KUKA KRL program: MyProgram_157().src

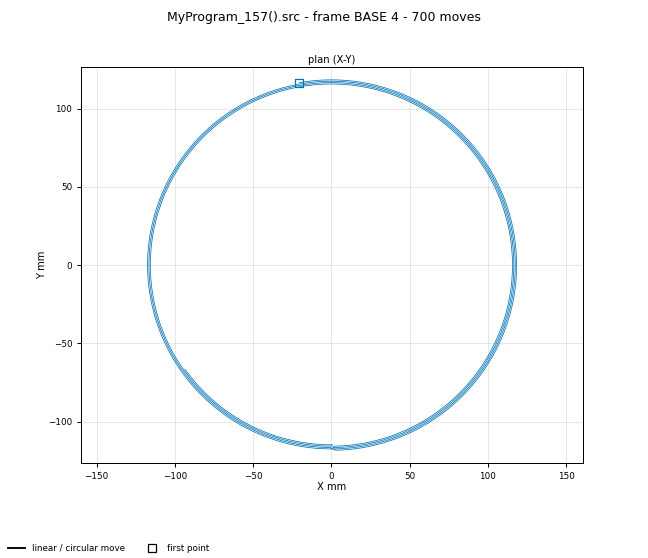
[picture p0: tool path of MyProgram_157().src in frame BASE 4, 700 of 700 moves have a stored position in this frame; points joined in program order, loops and branches not executed]
&ACCESS RVP
&REL 1
&PARAM TEMPLATE = C:\KRC\Roboter\Template\vorgabe
&PARAM EDITMASK = *
DEF MyProgram_157()
; ---- Setting reference (Base) ----
$BASE = BASE_DATA[4]

; --------------------------
; ---- Setting tool (TCP) ----
$TOOL = TOOL_DATA[3]
; --------------------------

$VEL.CP = VEL_APROX_PRINT
Startdeposition()
$VEL.CP = VEL_PRINT
LIN {X -20.7298,Y 116.5177,Z 121,A 95.4648,B 24.939,C -1.8039,E1 24.9731,E2 350.5826} C_DIS
LIN {X -17.3655,Y 117.0684,Z 121,A 93.8121,B 24.939,C -1.8049,E1 24.9777,E2 352.2344} C_DIS
LIN {X -14.6611,Y 117.4368,Z 121,A 92.4805,B 24.939,C -1.8053,E1 24.9814,E2 353.566} C_DIS
LIN {X -10.6565,Y 117.8666,Z 121,A 90.5367,B 24.9388,C -1.8066,E1 24.9868,E2 355.5079} C_DIS
LIN {X -7.2573,Y 118.1266,Z 121,A 88.8847,B 24.9388,C -1.8072,E1 24.9914,E2 357.1591} C_DIS
LIN {X -3.4087,Y 118.2982,Z 121,A 86.9833,B 24.9388,C -1.8062,E1 24.9967,E2 359.0632} C_DIS
LIN {X 0,Y 118.3494,Z 121,A 85.3671,B 24.9388,C -1.8081,E1 25.0012,E2 360.675} C_DIS
LIN {X 2.9044,Y 118.3137,Z 121,A 83.9605,B 24.9388,C -1.8082,E1 25.0051,E2 362.0809} C_DIS
LIN {X 5.8071,Y 118.2068,Z 121,A 82.5537,B 24.9388,C -1.8082,E1 25.009,E2 363.4872} C_DIS
LIN {X 9.9086,Y 117.9326,Z 121,A 80.5481,B 24.9388,C -1.8075,E1 25.0146,E2 365.4936} C_DIS
LIN {X 13.0447,Y 117.6283,Z 121,A 79.0389,B 24.9388,C -1.808,E1 25.0188,E2 367.0007} C_DIS
LIN {X 17.3655,Y 117.0684,Z 121,A 76.9308,B 24.9388,C -1.8076,E1 25.0246,E2 369.1081} C_DIS
LIN {X 21.1661,Y 116.4392,Z 121,A 75.01,B 24.939,C -1.8044,E1 25.0299,E2 371.0343} C_DIS
LIN {X 23.9622,Y 115.896,Z 121,A 73.6209,B 24.939,C -1.8034,E1 25.0338,E2 372.4243} C_DIS
LIN {X 27.3456,Y 115.1468,Z 121,A 72.0133,B 24.9389,C -1.8056,E1 25.0381,E2 374.0244} C_DIS
LIN {X 29.8333,Y 114.5258,Z 121,A 70.7927,B 24.9389,C -1.8058,E1 25.0414,E2 375.2426} C_DIS
LIN {X 32.4772,Y 113.8039,Z 121,A 69.3918,B 24.9392,C -1.8015,E1 25.0452,E2 376.6514} C_DIS
LIN {X 35.2603,Y 112.9726,Z 121,A 67.9878,B 24.9392,C -1.8006,E1 25.0489,E2 378.0551} C_DIS
LIN {X 39.3665,Y 111.608,Z 121,A 65.8909,B 24.9394,C -1.7987,E1 25.0545,E2 380.1524} C_DIS
LIN {X 43.4755,Y 110.0726,Z 121,A 63.8342,B 24.9393,C -1.7996,E1 25.0598,E2 382.2023} C_DIS
LIN {X 46.6287,Y 108.7765,Z 121,A 62.1876,B 24.9394,C -1.798,E1 25.0641,E2 383.8489} C_DIS
LIN {X 49.2842,Y 107.5995,Z 121,A 60.785,B 24.9395,C -1.7965,E1 25.0676,E2 385.2516} C_DIS
LIN {X 52.7592,Y 105.9366,Z 121,A 58.8678,B 24.9398,C -1.7919,E1 25.0725,E2 387.1747} C_DIS
LIN {X 55.7895,Y 104.3748,Z 121,A 57.2788,B 24.9398,C -1.7924,E1 25.0764,E2 388.7579} C_DIS
LIN {X 58.3342,Y 102.9742,Z 121,A 55.877,B 24.9399,C -1.7907,E1 25.0798,E2 390.1599} C_DIS
LIN {X 61.6537,Y 101.0194,Z 121,A 53.9611,B 24.9402,C -1.7855,E1 25.0844,E2 392.0819} C_DIS
LIN {X 64.5389,Y 99.2034,Z 121,A 52.373,B 24.9402,C -1.7858,E1 25.0881,E2 393.6643} C_DIS
LIN {X 67.7323,Y 97.0486,Z 121,A 50.4575,B 24.9406,C -1.7804,E1 25.0926,E2 395.5861} C_DIS
LIN {X 70.303,Y 95.2038,Z 121,A 48.9728,B 24.9406,C -1.7798,E1 25.0959,E2 397.0667} C_DIS
LIN {X 72.8123,Y 93.3003,Z 121,A 47.4695,B 24.9407,C -1.778,E1 25.0992,E2 398.5688} C_DIS
LIN {X 76.1971,Y 90.5571,Z 121,A 45.3689,B 24.941,C -1.7744,E1 25.1038,E2 400.6701} C_DIS
LIN {X 78.3965,Y 88.6598,Z 121,A 43.9683,B 24.9412,C -1.7719,E1 25.1067,E2 402.0711} C_DIS
LIN {X 81.2392,Y 86.0598,Z 121,A 42.1113,B 24.9414,C -1.7684,E1 25.1105,E2 403.9286} C_DIS
LIN {X 83.6856,Y 83.6856,Z 121,A 40.4685,B 24.9416,C -1.7652,E1 25.1138,E2 405.5722} C_DIS
LIN {X 85.7142,Y 81.6067,Z 121,A 39.069,B 24.9418,C -1.7624,E1 25.1165,E2 406.9722} C_DIS
LIN {X 88.6598,Y 78.3965,Z 121,A 36.9698,B 24.9421,C -1.7581,E1 25.1205,E2 409.0723} C_DIS
LIN {X 91.4853,Y 75.08,Z 121,A 34.8712,B 24.9424,C -1.7536,E1 25.1242,E2 411.1719} C_DIS
LIN {X 94.1868,Y 71.6618,Z 121,A 32.7728,B 24.9427,C -1.749,E1 25.1278,E2 413.2714} C_DIS
LIN {X 95.9171,Y 69.3288,Z 121,A 31.3738,B 24.9429,C -1.7458,E1 25.1302,E2 414.6712} C_DIS
LIN {X 97.5896,Y 66.954,Z 121,A 29.9754,B 24.9431,C -1.7426,E1 25.1324,E2 416.0703} C_DIS
LIN {X 99.2034,Y 64.5389,Z 121,A 28.577,B 24.9433,C -1.7393,E1 25.1345,E2 417.4695} C_DIS
LIN {X 100.7574,Y 62.0849,Z 121,A 27.1786,B 24.9435,C -1.7359,E1 25.1366,E2 418.8687} C_DIS
LIN {X 101.9939,Y 60.0278,Z 121,A 25.9667,B 24.9439,C -1.7304,E1 25.1384,E2 420.0873} C_DIS
LIN {X 103.6823,Y 57.0661,Z 121,A 24.3826,B 24.9439,C -1.729,E1 25.1405,E2 421.6666} C_DIS
LIN {X 105.0516,Y 54.5045,Z 121,A 22.9846,B 24.9442,C -1.7255,E1 25.1423,E2 423.0656} C_DIS
LIN {X 106.7681,Y 51.0556,Z 121,A 21.1306,B 24.9445,C -1.7208,E1 25.1446,E2 424.9207} C_DIS
LIN {X 107.9889,Y 48.42,Z 121,A 19.6765,B 24.9449,C -1.7144,E1 25.1463,E2 426.3819} C_DIS
LIN {X 109.3406,Y 45.2903,Z 121,A 18.0929,B 24.945,C -1.7128,E1 25.148,E2 427.9607} C_DIS
LIN {X 110.4191,Y 42.5933,Z 121,A 16.6957,B 24.9453,C -1.709,E1 25.1495,E2 429.359} C_DIS
LIN {X 111.745,Y 38.9763,Z 121,A 14.7858,B 24.9458,C -1.7013,E1 25.1513,E2 431.2764} C_DIS
LIN {X 112.8232,Y 35.7422,Z 121,A 13.2026,B 24.9458,C -1.6995,E1 25.1526,E2 432.8549} C_DIS
LIN {X 113.6663,Y 32.9626,Z 121,A 11.8056,B 24.9461,C -1.6956,E1 25.1537,E2 434.253} C_DIS
LIN {X 114.4411,Y 30.1632,Z 121,A 10.4084,B 24.9464,C -1.6917,E1 25.1548,E2 435.6515} C_DIS
LIN {X 115.1468,Y 27.3456,Z 121,A 9.0115,B 24.9466,C -1.6878,E1 25.1557,E2 437.0495} C_DIS
LIN {X 116.0753,Y 23.0888,Z 121,A 6.9164,B 24.947,C -1.6818,E1 25.1569,E2 439.1465} C_DIS
LIN {X 116.7633,Y 19.2984,Z 121,A 5.0071,B 24.9475,C -1.6738,E1 25.1578,E2 441.0635} C_DIS
LIN {X 117.2017,Y 16.4271,Z 121,A 3.6104,B 24.9478,C -1.6698,E1 25.1584,E2 442.4615} C_DIS
LIN {X 117.5901,Y 13.3702,Z 121,A 2.205,B 24.9478,C -1.6691,E1 25.1589,E2 443.8601} C_DIS
LIN {X 117.8666,Y 10.6565,Z 121,A 0.8739,B 24.9481,C -1.6644,E1 25.1592,E2 445.1945} C_DIS
LIN {X 118.1266,Y 7.2573,Z 121,A -0.7652,B 24.9484,C -1.6595,E1 25.1595,E2 446.8353} C_DIS
LIN {X 118.2982,Y 3.4087,Z 121,A -2.674,B 24.9489,C -1.6514,E1 25.1597,E2 448.7519} C_DIS
LIN {X 118.3493,Y 0,Z 121,A -4.4183,B 24.9495,C -1.6414,E1 25.1597,E2 450.5093} C_DIS
LIN {X 118.2847,Y -3.8518,Z 121,A -6.1653,B 24.9495,C -1.6411,E1 25.1597,E2 452.2467} C_DIS
LIN {X 118.1266,Y -7.2573,Z 121,A -7.7477,B 24.9497,C -1.6389,E1 25.1594,E2 453.8248} C_DIS
LIN {X 117.913,Y -10.1541,Z 121,A -9.1441,B 24.9499,C -1.6348,E1 25.1591,E2 455.2227} C_DIS
LIN {X 117.6283,Y -13.0447,Z 121,A -10.5406,B 24.9502,C -1.6307,E1 25.1587,E2 456.6206} C_DIS
LIN {X 117.0684,Y -17.3655,Z 121,A -12.6352,B 24.9506,C -1.6245,E1 25.1579,E2 458.7174} C_DIS
LIN {X 116.607,Y -20.2332,Z 121,A -14.0318,B 24.9508,C -1.6204,E1 25.1573,E2 460.1155} C_DIS
LIN {X 116.0753,Y -23.0888,Z 121,A -15.4284,B 24.951,C -1.6163,E1 25.1565,E2 461.5137} C_DIS
LIN {X 115.4737,Y -25.9305,Z 121,A -16.825,B 24.9513,C -1.6122,E1 25.1557,E2 462.9117} C_DIS
LIN {X 114.5667,Y -29.6745,Z 121,A -18.6774,B 24.9516,C -1.6068,E1 25.1545,E2 464.766} C_DIS
LIN {X 113.8039,Y -32.4772,Z 121,A -20.1306,B 24.952,C -1.6001,E1 25.1534,E2 466.2269} C_DIS
LIN {X 112.9726,Y -35.2603,Z 121,A -21.5273,B 24.9523,C -1.596,E1 25.1522,E2 467.6251} C_DIS
LIN {X 111.5982,Y -39.3946,Z 121,A -23.6224,B 24.9526,C -1.5901,E1 25.1503,E2 469.7225} C_DIS
LIN {X 110.4191,Y -42.5933,Z 121,A -25.2053,B 24.9527,C -1.5881,E1 25.1488,E2 471.3012} C_DIS
LIN {X 108.7765,Y -46.6287,Z 121,A -27.3008,B 24.9531,C -1.5822,E1 25.1466,E2 473.399} C_DIS
LIN {X 107.8067,Y -48.8242,Z 121,A -28.5117,B 24.9534,C -1.5763,E1 25.1452,E2 474.6172} C_DIS
LIN {X 106.3576,Y -51.91,Z 121,A -30.0949,B 24.9535,C -1.5745,E1 25.1433,E2 476.1962} C_DIS
LIN {X 105.0871,Y -54.4349,Z 121,A -31.4564,B 24.9538,C -1.5708,E1 25.1415,E2 477.5593} C_DIS
LIN {X 103.6823,Y -57.0661,Z 121,A -32.8894,B 24.954,C -1.567,E1 25.1396,E2 478.9938} C_DIS
LIN {X 102.2506,Y -59.5934,Z 121,A -34.287,B 24.9542,C -1.5633,E1 25.1377,E2 480.3928} C_DIS
LIN {X 100.7573,Y -62.0849,Z 121,A -35.6846,B 24.9544,C -1.5596,E1 25.1356,E2 481.792} C_DIS
LIN {X 98.4039,Y -65.7514,Z 121,A -37.7809,B 24.9547,C -1.5542,E1 25.1325,E2 483.8906} C_DIS
LIN {X 96.2101,Y -68.9181,Z 121,A -39.6351,B 24.955,C -1.5495,E1 25.1295,E2 485.7467} C_DIS
LIN {X 94.5528,Y -71.1746,Z 121,A -41.0138,B 24.9553,C -1.5447,E1 25.1272,E2 487.1302} C_DIS
LIN {X 92.3998,Y -73.9517,Z 121,A -42.6739,B 24.9555,C -1.542,E1 25.1243,E2 488.7889} C_DIS
LIN {X 90.5571,Y -76.1971,Z 121,A -44.0724,B 24.9556,C -1.5386,E1 25.1218,E2 490.1888} C_DIS
LIN {X 88.6598,Y -78.3965,Z 121,A -45.4709,B 24.9558,C -1.5353,E1 25.1192,E2 491.5889} C_DIS
LIN {X 86.069,Y -81.2294,Z 121,A -47.3786,B 24.9562,C -1.5283,E1 25.1156,E2 493.5048} C_DIS
LIN {X 83.6856,Y -83.6856,Z 121,A -48.9679,B 24.9562,C -1.5273,E1 25.1125,E2 495.0895} C_DIS
LIN {X 80.9162,Y -86.3635,Z 121,A -50.8798,B 24.9567,C -1.5206,E1 25.1086,E2 497.0094} C_DIS
LIN {X 77.6826,Y -89.2833,Z 121,A -52.9786,B 24.9569,C -1.5162,E1 25.1042,E2 499.1102} C_DIS
LIN {X 74.3437,Y -92.0821,Z 121,A -55.0212,B 24.957,C -1.5146,E1 25.0999,E2 501.1488} C_DIS
LIN {X 72.0615,Y -93.8788,Z 121,A -56.4774,B 24.9573,C -1.5091,E1 25.0966,E2 502.6125} C_DIS
LIN {X 69.3288,Y -95.9171,Z 121,A -58.0641,B 24.9573,C -1.5086,E1 25.0931,E2 504.1947} C_DIS
LIN {X 66.954,Y -97.5896,Z 121,A -59.4641,B 24.9575,C -1.506,E1 25.0899,E2 505.5961} C_DIS
LIN {X 64.9601,Y -98.9256,Z 121,A -60.6777,B 24.9578,C -1.5013,E1 25.087,E2 506.8168} C_DIS
LIN {X 62.0849,Y -100.7573,Z 121,A -62.2646,B 24.9578,C -1.5011,E1 25.0833,E2 508.3991} C_DIS
LIN {X 59.5934,Y -102.2506,Z 121,A -63.6655,B 24.9579,C -1.4987,E1 25.0799,E2 509.8013} C_DIS
LIN {X 56.233,Y -104.1343,Z 121,A -65.4978,B 24.958,C -1.497,E1 25.0754,E2 511.6324} C_DIS
LIN {X 53.6605,Y -105.4829,Z 121,A -66.9246,B 24.9582,C -1.4936,E1 25.0719,E2 513.0632} C_DIS
LIN {X 51.0556,Y -106.7681,Z 121,A -68.3222,B 24.9583,C -1.4917,E1 25.0684,E2 514.4616} C_DIS
LIN {X 47.9601,Y -108.1961,Z 121,A -69.9709,B 24.9585,C -1.4892,E1 25.0642,E2 516.1122} C_DIS
LIN {X 43.9452,Y -109.8881,Z 121,A -72.0737,B 24.9586,C -1.4864,E1 25.0587,E2 518.2167} C_DIS
LIN {X 40.3447,Y -111.2583,Z 121,A -73.9903,B 24.9589,C -1.4815,E1 25.0537,E2 520.1408} C_DIS
LIN {X 36.2222,Y -112.6678,Z 121,A -76.0939,B 24.959,C -1.4791,E1 25.0481,E2 522.246} C_DIS
LIN {X 33.4463,Y -113.5229,Z 121,A -77.4966,B 24.959,C -1.4777,E1 25.0444,E2 523.6497} C_DIS
LIN {X 30.1632,Y -114.4411,Z 121,A -79.0867,B 24.959,C -1.4786,E1 25.0401,E2 525.2349} C_DIS
LIN {X 26.4221,Y -115.3602,Z 121,A -80.9477,B 24.9591,C -1.477,E1 25.0351,E2 527.0971} C_DIS
LIN {X 23.0888,Y -116.0753,Z 121,A -82.5949,B 24.9592,C -1.4757,E1 25.0306,E2 528.7454} C_DIS
LIN {X 19.2984,Y -116.7633,Z 121,A -84.5139,B 24.9594,C -1.4717,E1 25.0253,E2 530.6717} C_DIS
LIN {X 16.4271,Y -117.2017,Z 121,A -85.9181,B 24.9594,C -1.4708,E1 25.0214,E2 532.0767} C_DIS
LIN {X 13.0447,Y -117.6283,Z 121,A -87.5095,B 24.9594,C -1.4725,E1 25.017,E2 533.663} C_DIS
LIN {X 10.1541,Y -117.913,Z 121,A -88.9137,B 24.9594,C -1.4718,E1 25.0131,E2 535.0679} C_DIS
LIN {X 7.2573,Y -118.1266,Z 121,A -90.3189,B 24.9594,C -1.4712,E1 25.0092,E2 536.4739} C_DIS
LIN {X 2.9044,Y -118.3137,Z 121,A -92.4266,B 24.9594,C -1.4706,E1 25.0033,E2 538.5826} C_DIS
LIN {X 2.9044,Y -118.3137,Z 121,A -92.4266,B 24.9594,C -1.4706,E1 25.0033,E2 538.5826} C_DIS
Enddeposition()
LIN {X 0.8321,Y -117.4596,Z 121,A -93.3395,B 24.9584,C -1.49,E1 25.0009,E2 539.4494} C_DIS
Startdeposition()
$VEL.CP = VEL_PRINT
LIN {X 3.2999,Y -117.4195,Z 121,A -91.5559,B 24.9569,C -1.5166,E1 25.006,E2 537.603} C_DIS
LIN {X 6.8139,Y -117.2681,Z 121,A -89.8243,B 24.9569,C -1.518,E1 25.0108,E2 535.8686} C_DIS
LIN {X 10.3893,Y -117.0058,Z 121,A -88.0253,B 24.9566,C -1.5212,E1 25.0159,E2 534.0631} C_DIS
LIN {X 14.3068,Y -116.5927,Z 121,A -86.0792,B 24.9566,C -1.5235,E1 25.0213,E2 532.1131} C_DIS
LIN {X 17.0501,Y -116.2227,Z 121,A -84.8996,B 24.9569,C -1.5166,E1 25.0245,E2 530.9508} C_DIS
LIN {X 21.5545,Y -115.4729,Z 121,A -82.5382,B 24.9565,C -1.5245,E1 25.031,E2 528.5731} C_DIS
LIN {X 24.947,Y -114.7858,Z 121,A -80.9226,B 24.9565,C -1.5227,E1 25.0354,E2 526.964} C_DIS
LIN {X 27.5735,Y -114.1837,Z 121,A -79.0122,B 24.9549,C -1.5518,E1 25.0408,E2 524.9874} C_DIS
LIN {X 31.8685,Y -113.06,Z 121,A -77.3966,B 24.9562,C -1.5284,E1 25.045,E2 523.4297} C_DIS
LIN {X 36.1496,Y -111.7647,Z 121,A -75.3333,B 24.9564,C -1.5255,E1 25.0505,E2 521.3772} C_DIS
LIN {X 39.0961,Y -110.7685,Z 121,A -73.7738,B 24.9562,C -1.5294,E1 25.0546,E2 519.8115} C_DIS
LIN {X 43.4706,Y -109.1272,Z 121,A -71.4393,B 24.9558,C -1.5351,E1 25.0607,E2 517.4685} C_DIS
LIN {X 46.5849,Y -107.8338,Z 121,A -69.8145,B 24.9558,C -1.5366,E1 25.0649,E2 515.844} C_DIS
LIN {X 49.5604,Y -106.4984,Z 121,A -68.2686,B 24.9558,C -1.537,E1 25.0688,E2 514.301} C_DIS
LIN {X 53.0811,Y -104.7889,Z 121,A -66.5543,B 24.9561,C -1.531,E1 25.073,E2 512.6055} C_DIS
LIN {X 56.616,Y -102.9234,Z 121,A -64.3099,B 24.9551,C -1.5483,E1 25.0786,E2 510.3266} C_DIS
LIN {X 59.527,Y -101.2657,Z 121,A -62.7876,B 24.9552,C -1.546,E1 25.0823,E2 508.8144} C_DIS
LIN {X 62.3026,Y -99.5818,Z 121,A -61.1934,B 24.955,C -1.5496,E1 25.0861,E2 507.2167} C_DIS
LIN {X 65.7863,Y -97.3155,Z 121,A -59.2186,B 24.955,C -1.5511,E1 25.0907,E2 505.2449} C_DIS
LIN {X 68.4047,Y -95.4933,Z 121,A -57.8037,B 24.9551,C -1.5477,E1 25.0939,E2 503.8431} C_DIS
LIN {X 72.3765,Y -92.5208,Z 121,A -54.5882,B 24.9526,C -1.591,E1 25.1012,E2 500.5371} C_DIS
LIN {X 75.9705,Y -89.5918,Z 121,A -52.9888,B 24.9542,C -1.5643,E1 25.1045,E2 499.0069} C_DIS
LIN {X 79.7422,Y -86.2515,Z 121,A -50.3792,B 24.9534,C -1.5774,E1 25.1099,E2 496.3768} C_DIS
LIN {X 83.2682,Y -82.8525,Z 121,A -47.8356,B 24.9526,C -1.5907,E1 25.115,E2 493.8125} C_DIS
LIN {X 85.5139,Y -80.5327,Z 121,A -46.7222,B 24.9537,C -1.5725,E1 25.1171,E2 492.7469} C_DIS
LIN {X 88.3698,Y -77.3882,Z 121,A -44.5319,B 24.953,C -1.5835,E1 25.1212,E2 490.5404} C_DIS
LIN {X 90.7856,Y -74.5426,Z 121,A -42.7886,B 24.953,C -1.5845,E1 25.1243,E2 488.8026} C_DIS
LIN {X 92.9303,Y -71.848,Z 121,A -41.0839,B 24.9526,C -1.5903,E1 25.1272,E2 487.0923} C_DIS
LIN {X 94.8498,Y -69.2941,Z 121,A -39.5118,B 24.9523,C -1.5953,E1 25.1299,E2 485.516} C_DIS
LIN {X 97.0567,Y -66.1684,Z 121,A -37.7561,B 24.9523,C -1.5952,E1 25.1326,E2 483.7692} C_DIS
LIN {X 98.672,Y -63.7345,Z 121,A -36.434,B 24.9523,C -1.5943,E1 25.1347,E2 482.4557} C_DIS
LIN {X 100.7204,Y -60.448,Z 121,A -34.2239,B 24.9511,C -1.6153,E1 25.1379,E2 480.2075} C_DIS
LIN {X 102.8049,Y -56.829,Z 121,A -32.2704,B 24.951,C -1.6172,E1 25.1406,E2 478.2595} C_DIS
LIN {X 104.4904,Y -53.6651,Z 121,A -30.6953,B 24.9512,C -1.6141,E1 25.1426,E2 476.7001} C_DIS
LIN {X 105.8226,Y -50.9876,Z 121,A -29.2209,B 24.9509,C -1.6193,E1 25.1444,E2 475.2214} C_DIS
LIN {X 107.3121,Y -47.7758,Z 121,A -27.3557,B 24.9501,C -1.6312,E1 25.1466,E2 473.3381} C_DIS
LIN {X 108.8767,Y -44.0914,Z 121,A -25.4954,B 24.9501,C -1.6328,E1 25.1486,E2 471.4843} C_DIS
LIN {X 110.3331,Y -40.3081,Z 121,A -23.5273,B 24.9497,C -1.6386,E1 25.1505,E2 469.5135} C_DIS
LIN {X 112.5098,Y -33.7612,Z 121,A -20.1836,B 24.9491,C -1.6482,E1 25.1534,E2 466.1663} C_DIS
LIN {X 113.818,Y -29.0452,Z 121,A -17.8234,B 24.9487,C -1.6545,E1 25.1551,E2 463.8046} C_DIS
LIN {X 114.7059,Y -25.3135,Z 121,A -15.9774,B 24.9484,C -1.6593,E1 25.1563,E2 461.958} C_DIS
LIN {X 115.4119,Y -21.8711,Z 121,A -14.3015,B 24.9482,C -1.663,E1 25.1572,E2 460.2832} C_DIS
LIN {X 115.9573,Y -18.7721,Z 121,A -12.6525,B 24.9475,C -1.6736,E1 25.158,E2 458.619} C_DIS
LIN {X 116.5771,Y -14.4341,Z 121,A -10.4812,B 24.947,C -1.6822,E1 25.1588,E2 456.4402} C_DIS
LIN {X 116.9803,Y -10.6656,Z 121,A -8.7611,B 24.947,C -1.682,E1 25.1592,E2 454.7308} C_DIS
LIN {X 117.2798,Y -6.603,Z 121,A -6.7288,B 24.9464,C -1.6907,E1 25.1596,E2 452.6899} C_DIS
LIN {X 117.4395,Y -2.4929,Z 121,A -4.8179,B 24.9464,C -1.6926,E1 25.1598,E2 450.7859} C_DIS
LIN {X 117.4621,Y 0.9671,Z 121,A -3.0388,B 24.9457,C -1.7026,E1 25.1598,E2 448.994} C_DIS
LIN {X 117.3604,Y 4.967,Z 121,A -1.1861,B 24.9456,C -1.7041,E1 25.1596,E2 447.1487} C_DIS
LIN {X 117.1297,Y 8.8879,Z 121,A 0.6551,B 24.9454,C -1.7067,E1 25.1592,E2 445.3123} C_DIS
LIN {X 116.8294,Y 12.2075,Z 121,A 2.3671,B 24.9448,C -1.7161,E1 25.1588,E2 443.5882} C_DIS
LIN {X 116.3353,Y 16.2574,Z 121,A 4.3009,B 24.9446,C -1.7198,E1 25.1581,E2 441.6572} C_DIS
LIN {X 115.8422,Y 19.4608,Z 121,A 5.83,B 24.9444,C -1.7223,E1 25.1574,E2 440.1311} C_DIS
LIN {X 115.2313,Y 22.8093,Z 121,A 7.8143,B 24.943,C -1.7432,E1 25.1563,E2 438.1091} C_DIS
LIN {X 114.1359,Y 27.7692,Z 121,A 9.9681,B 24.9436,C -1.7353,E1 25.155,E2 435.9864} C_DIS
LIN {X 113.2965,Y 31.0193,Z 121,A 11.5935,B 24.9433,C -1.7398,E1 25.1538,E2 434.3598} C_DIS
LIN {X 112.537,Y 33.6693,Z 121,A 13.2708,B 24.9419,C -1.76,E1 25.1525,E2 432.6443} C_DIS
LIN {X 111.5369,Y 36.8533,Z 121,A 14.6663,B 24.9424,C -1.7537,E1 25.1513,E2 431.2717} C_DIS
LIN {X 110.3661,Y 40.2178,Z 121,A 16.2948,B 24.9424,C -1.7537,E1 25.1497,E2 429.6524} C_DIS
LIN {X 108.9824,Y 43.8315,Z 121,A 18.1047,B 24.9422,C -1.7555,E1 25.1479,E2 427.8482} C_DIS
LIN {X 107.6921,Y 46.91,Z 121,A 19.6476,B 24.9422,C -1.7562,E1 25.1462,E2 426.3122} C_DIS
LIN {X 106.1333,Y 50.3408,Z 121,A 22.3438,B 24.9391,C -1.8028,E1 25.1429,E2 423.5204} C_DIS
LIN {X 103.8916,Y 54.815,Z 121,A 24.0413,B 24.941,C -1.7738,E1 25.1408,E2 421.9004} C_DIS
LIN {X 102.0703,Y 58.1377,Z 121,A 25.8931,B 24.9407,C -1.779,E1 25.1383,E2 420.0459} C_DIS
LIN {X 100.5204,Y 60.777,Z 121,A 27.2357,B 24.9409,C -1.7759,E1 25.1364,E2 418.7176} C_DIS
LIN {X 98.6915,Y 63.7041,Z 121,A 29.5071,B 24.9387,C -1.8085,E1 25.1329,E2 416.3808} C_DIS
LIN {X 96.5397,Y 66.9196,Z 121,A 31.326,B 24.9386,C -1.81,E1 25.13,E2 414.5671} C_DIS
LIN {X 94.3656,Y 69.9551,Z 121,A 32.6495,B 24.9399,C -1.7908,E1 25.1279,E2 413.2954} C_DIS
LIN {X 92.4451,Y 72.4724,Z 121,A 34.2293,B 24.9395,C -1.7963,E1 25.1252,E2 411.7102} C_DIS
LIN {X 90.7782,Y 74.5514,Z 121,A 35.6238,B 24.939,C -1.8039,E1 25.1227,E2 410.3042} C_DIS
LIN {X 88.4019,Y 77.3515,Z 121,A 37.3344,B 24.939,C -1.8043,E1 25.1196,E2 408.6004} C_DIS
LIN {X 85.9021,Y 80.1199,Z 121,A 39.2627,B 24.9384,C -1.8135,E1 25.1159,E2 406.6587} C_DIS
LIN {X 82.9142,Y 83.2084,Z 121,A 41.2151,B 24.9385,C -1.8113,E1 25.1121,E2 404.7199} C_DIS
LIN {X 80.6743,Y 85.3807,Z 121,A 42.7029,B 24.9384,C -1.8129,E1 25.1091,E2 403.2344} C_DIS
LIN {X 78.2297,Y 87.6258,Z 121,A 44.343,B 24.9381,C -1.8172,E1 25.1057,E2 401.5908} C_DIS
LIN {X 75.253,Y 90.1952,Z 121,A 46.9929,B 24.9355,C -1.8554,E1 25.0999,E2 398.8607} C_DIS
LIN {X 71.2921,Y 93.3586,Z 121,A 48.8424,B 24.9372,C -1.8306,E1 25.0959,E2 397.0768} C_DIS
LIN {X 68.8181,Y 95.1982,Z 121,A 50.3454,B 24.937,C -1.8332,E1 25.0926,E2 395.573} C_DIS
LIN {X 66.325,Y 96.9508,Z 121,A 51.7855,B 24.937,C -1.8335,E1 25.0892,E2 394.137} C_DIS
LIN {X 63.5754,Y 98.7741,Z 121,A 53.1884,B 24.9375,C -1.8265,E1 25.086,E2 392.7552} C_DIS
LIN {X 61.2629,Y 100.2251,Z 121,A 54.5665,B 24.9372,C -1.8308,E1 25.0827,E2 391.3715} C_DIS
LIN {X 58.2969,Y 101.9788,Z 121,A 56.3672,B 24.9366,C -1.8388,E1 25.0783,E2 389.5572} C_DIS
LIN {X 54.7673,Y 103.9167,Z 121,A 58.3102,B 24.9366,C -1.8405,E1 25.0736,E2 387.6157} C_DIS
LIN {X 51.2509,Y 105.696,Z 121,A 60.2593,B 24.9363,C -1.8442,E1 25.0687,E2 385.6632} C_DIS
LIN {X 47.6547,Y 107.3667,Z 121,A 62.1737,B 24.9362,C -1.8455,E1 25.0638,E2 383.7505} C_DIS
LIN {X 44.4763,Y 108.72,Z 121,A 63.8325,B 24.9362,C -1.8461,E1 25.0596,E2 382.0941} C_DIS
LIN {X 40.8745,Y 110.1265,Z 121,A 65.7701,B 24.9358,C -1.8503,E1 25.0545,E2 380.1508} C_DIS
LIN {X 37.3056,Y 111.3844,Z 121,A 68.0183,B 24.9344,C -1.8703,E1 25.0484,E2 377.8594} C_DIS
LIN {X 33.5434,Y 112.5744,Z 121,A 69.8704,B 24.9346,C -1.8684,E1 25.0435,E2 376.0151} C_DIS
LIN {X 29.9249,Y 113.5918,Z 121,A 71.2033,B 24.9361,C -1.8468,E1 25.04,E2 374.7356} C_DIS
LIN {X 26.9203,Y 114.3402,Z 121,A 72.8671,B 24.9355,C -1.8546,E1 25.0355,E2 373.0557} C_DIS
LIN {X 23.1374,Y 115.1653,Z 121,A 74.7881,B 24.9354,C -1.857,E1 25.0302,E2 371.1314} C_DIS
LIN {X 19.1105,Y 115.9008,Z 121,A 76.6553,B 24.9357,C -1.8519,E1 25.0251,E2 369.2784} C_DIS
LIN {X 15.7309,Y 116.4091,Z 121,A 78.2397,B 24.9359,C -1.8486,E1 25.0208,E2 367.7031} C_DIS
LIN {X 12.4103,Y 116.8082,Z 121,A 79.9364,B 24.9357,C -1.8518,E1 25.016,E2 365.9999} C_DIS
LIN {X 9.0609,Y 117.1159,Z 121,A 81.691,B 24.9354,C -1.8571,E1 25.0111,E2 364.2339} C_DIS
LIN {X 5.751,Y 117.3267,Z 121,A 83.3791,B 24.9351,C -1.8601,E1 25.0064,E2 362.5391} C_DIS
LIN {X 1.4546,Y 117.4582,Z 121,A 85.3149,B 24.9357,C -1.8527,E1 25.001,E2 360.6213} C_DIS
LIN {X -1.9991,Y 117.4486,Z 121,A 87.0648,B 24.9355,C -1.8553,E1 24.9961,E2 358.8653} C_DIS
LIN {X -6.0792,Y 117.3087,Z 121,A 88.8438,B 24.9362,C -1.8452,E1 24.9912,E2 357.1098} C_DIS
LIN {X -8.9147,Y 117.1275,Z 121,A 90.2049,B 24.9362,C -1.8435,E1 24.9875,E2 355.7522} C_DIS
LIN {X -12.0639,Y 116.8444,Z 121,A 91.9415,B 24.9358,C -1.8513,E1 24.9826,E2 353.9961} C_DIS
LIN {X -15.7391,Y 116.4081,Z 121,A 93.8439,B 24.9355,C -1.8545,E1 24.9773,E2 352.0849} C_DIS
LIN {X -19.8135,Y 115.7832,Z 121,A 95.9275,B 24.9355,C -1.8562,E1 24.9715,E2 349.9951} C_DIS
LIN {X -27.3101,Y 114.2476,Z 121,A 99.7512,B 24.9354,C -1.8569,E1 24.9611,E2 346.1651} C_DIS
LIN {X -32.0342,Y 113.013,Z 121,A 101.8923,B 24.9363,C -1.8439,E1 24.9554,E2 344.0515} C_DIS
LIN {X -35.7831,Y 111.8832,Z 121,A 103.8824,B 24.9362,C -1.8452,E1 24.9501,E2 342.055} C_DIS
LIN {X -39.636,Y 110.5783,Z 121,A 105.7936,B 24.9366,C -1.8395,E1 24.945,E2 340.1535} C_DIS
LIN {X -43.2643,Y 109.2083,Z 121,A 107.6527,B 24.9368,C -1.8356,E1 24.9402,E2 338.2999} C_DIS
LIN {X -50.1091,Y 106.243,Z 121,A 111.442,B 24.9368,C -1.8365,E1 24.9305,E2 334.4992} C_DIS
LIN {X -52.5867,Y 105.0381,Z 121,A 112.9317,B 24.9365,C -1.8406,E1 24.9268,E2 332.9958} C_DIS
LIN {X -56.8256,Y 102.8068,Z 121,A 115.0146,B 24.9375,C -1.8257,E1 24.9217,E2 330.9425} C_DIS
LIN {X -59.2175,Y 101.4487,Z 121,A 116.4587,B 24.9374,C -1.8277,E1 24.9182,E2 329.4895} C_DIS
LIN {X -62.1676,Y 99.6661,Z 121,A 117.9064,B 24.9383,C -1.8146,E1 24.9148,E2 328.0684} C_DIS
LIN {X -64.0959,Y 98.4392,Z 121,A 119.288,B 24.9377,C -1.8238,E1 24.9115,E2 326.6604} C_DIS
LIN {X -68.4041,Y 95.4938,Z 121,A 121.8034,B 24.9381,C -1.8174,E1 24.9058,E2 324.1518} C_DIS
LIN {X -71.4545,Y 93.2335,Z 121,A 123.6221,B 24.9385,C -1.812,E1 24.9017,E2 322.3392} C_DIS
LIN {X -74.1517,Y 91.1028,Z 121,A 125.3091,B 24.9387,C -1.8088,E1 24.8981,E2 320.6536} C_DIS
LIN {X -77.1304,Y 88.595,Z 121,A 127.0055,B 24.9395,C -1.7959,E1 24.8945,E2 318.9812} C_DIS
LIN {X -79.3821,Y 86.583,Z 121,A 128.6575,B 24.9393,C -1.8,E1 24.891,E2 317.3128} C_DIS
LIN {X -82.1034,Y 84.0093,Z 121,A 130.5775,B 24.9393,C -1.7996,E1 24.8872,E2 315.386} C_DIS
LIN {X -84.7278,Y 81.3595,Z 121,A 132.3892,B 24.9396,C -1.7948,E1 24.8836,E2 313.5779} C_DIS
LIN {X -87.3955,Y 78.4869,Z 121,A 134.2484,B 24.9401,C -1.7877,E1 24.8802,E2 311.7273} C_DIS
LIN {X -89.7973,Y 75.7293,Z 121,A 136.0212,B 24.9404,C -1.7826,E1 24.8769,E2 309.9586} C_DIS
LIN {X -92.094,Y 72.9167,Z 121,A 137.7038,B 24.941,C -1.7742,E1 24.874,E2 308.2882} C_DIS
LIN {X -93.5149,Y 71.0883,Z 121,A 139.1211,B 24.9404,C -1.7831,E1 24.8716,E2 306.8428} C_DIS
LIN {X -95.6872,Y 68.1329,Z 121,A 140.7571,B 24.9412,C -1.7718,E1 24.8689,E2 305.2258} C_DIS
LIN {X -97.8621,Y 64.9713,Z 121,A 142.6397,B 24.9415,C -1.767,E1 24.866,E2 303.3453} C_DIS
LIN {X -99.5406,Y 62.3684,Z 121,A 144.1789,B 24.9417,C -1.7639,E1 24.8637,E2 301.8057} C_DIS
LIN {X -101.396,Y 59.3066,Z 121,A 146.0219,B 24.9417,C -1.7628,E1 24.861,E2 299.9557} C_DIS
LIN {X -103.6755,Y 55.2253,Z 121,A 148.2584,B 24.9423,C -1.7543,E1 24.8581,E2 297.7279} C_DIS
LIN {X -104.8636,Y 52.9348,Z 121,A 149.7413,B 24.942,C -1.7598,E1 24.8562,E2 296.2237} C_DIS
LIN {X -106.9367,Y 48.6088,Z 121,A 151.6356,B 24.9436,C -1.7343,E1 24.854,E2 294.3801} C_DIS
LIN {X -108.0879,Y 45.9925,Z 121,A 153.058,B 24.9438,C -1.7311,E1 24.8524,E2 292.9573} C_DIS
LIN {X -109.2054,Y 43.2716,Z 121,A 154.6453,B 24.9438,C -1.733,E1 24.8507,E2 291.3566} C_DIS
LIN {X -110.2298,Y 40.5914,Z 121,A 156.0709,B 24.9439,C -1.7297,E1 24.8493,E2 289.9309} C_DIS
LIN {X -111.4801,Y 37.0217,Z 121,A 158.1326,B 24.9437,C -1.7329,E1 24.8474,E2 287.8499} C_DIS
LIN {X -112.7909,Y 32.8137,Z 121,A 160.2245,B 24.9443,C -1.7237,E1 24.8458,E2 285.7679} C_DIS
LIN {X -114.6039,Y 25.7787,Z 121,A 163.7731,B 24.945,C -1.7124,E1 24.8434,E2 282.2253} C_DIS
LIN {X -115.3539,Y 22.1723,Z 121,A 165.3692,B 24.9459,C -1.6984,E1 24.8425,E2 280.6533} C_DIS
LIN {X -116.0063,Y 18.4644,Z 121,A 167.4636,B 24.9456,C -1.7031,E1 24.8415,E2 278.5353} C_DIS
LIN {X -116.5625,Y 14.5472,Z 121,A 169.2381,B 24.9465,C -1.6904,E1 24.8409,E2 276.7805} C_DIS
LIN {X -116.9389,Y 11.1147,Z 121,A 170.9896,B 24.9466,C -1.6877,E1 24.8404,E2 275.025} C_DIS
LIN {X -117.2413,Y 7.2822,Z 121,A 172.9883,B 24.9466,C -1.6866,E1 24.84,E2 273.0166} C_DIS
LIN {X -117.4349,Y 2.7421,Z 121,A 175.3055,B 24.9469,C -1.6836,E1 24.8398,E2 270.6928} C_DIS
LIN {X -117.4508,Y -1.8747,Z 121,A 177.3802,B 24.9478,C -1.6689,E1 24.8398,E2 268.6405} C_DIS
LIN {X -117.3633,Y -4.8994,Z 121,A 178.8763,B 24.9481,C -1.665,E1 24.84,E2 267.1449} C_DIS
LIN {X -117.1316,Y -8.8645,Z 121,A -179.1565,B 24.9484,C -1.6599,E1 24.8403,E2 265.1778} C_DIS
LIN {X -116.8302,Y -12.1999,Z 121,A -177.574,B 24.9488,C -1.6526,E1 24.8408,E2 263.6034} C_DIS
LIN {X -116.453,Y -15.3921,Z 121,A -176.112,B 24.9494,C -1.6432,E1 24.8413,E2 262.1551} C_DIS
LIN {X -115.7092,Y -20.244,Z 121,A -173.4721,B 24.9492,C -1.6457,E1 24.8425,E2 259.4935} C_DIS
LIN {X -114.6123,Y -25.7423,Z 121,A -170.7012,B 24.9497,C -1.6386,E1 24.844,E2 256.7232} C_DIS
LIN {X -113.8328,Y -28.9879,Z 121,A -169.2105,B 24.9503,C -1.6278,E1 24.845,E2 255.2494} C_DIS
LIN {X -113.1263,Y -31.6345,Z 121,A -167.8365,B 24.9505,C -1.6253,E1 24.846,E2 253.8734} C_DIS
LIN {X -112.1911,Y -34.8035,Z 121,A -166.194,B 24.9507,C -1.6217,E1 24.8474,E2 252.2302} C_DIS
LIN {X -110.9879,Y -38.471,Z 121,A -164.1531,B 24.9507,C -1.6226,E1 24.8492,E2 250.1754} C_DIS
LIN {X -109.5191,Y -42.4731,Z 121,A -162.354,B 24.9518,C -1.6047,E1 24.8509,E2 248.4089} C_DIS
LIN {X -108.6609,Y -44.6215,Z 121,A -160.7538,B 24.9508,C -1.6212,E1 24.8527,E2 246.7604} C_DIS
LIN {X -107.396,Y -47.5891,Z 121,A -159.361,B 24.9515,C -1.609,E1 24.8542,E2 245.389} C_DIS
LIN {X -105.5624,Y -51.5289,Z 121,A -157.2238,B 24.9518,C -1.6037,E1 24.8568,E2 243.2528} C_DIS
LIN {X -104.0752,Y -54.4664,Z 121,A -155.6677,B 24.9522,C -1.5971,E1 24.8588,E2 241.704} C_DIS
LIN {X -102.3643,Y -57.6181,Z 121,A -153.9344,B 24.9525,C -1.5917,E1 24.8611,E2 239.9747} C_DIS
LIN {X -100.4968,Y -60.816,Z 121,A -152.1361,B 24.9528,C -1.5865,E1 24.8637,E2 238.1794} C_DIS
LIN {X -98.7032,Y -63.6859,Z 121,A -150.4671,B 24.9531,C -1.5829,E1 24.8662,E2 236.5105} C_DIS
LIN {X -96.0864,Y -67.5718,Z 121,A -148.0928,B 24.9531,C -1.5808,E1 24.87,E2 234.1294} C_DIS
LIN {X -93.3646,Y -71.2843,Z 121,A -145.8212,B 24.9534,C -1.5764,E1 24.8738,E2 231.8574} C_DIS
LIN {X -90.7928,Y -74.5339,Z 121,A -143.7589,B 24.9536,C -1.5733,E1 24.8774,E2 229.7929} C_DIS
LIN {X -88.1642,Y -77.6236,Z 121,A -141.8114,B 24.954,C -1.5674,E1 24.8809,E2 227.8506} C_DIS
LIN {X -85.4616,Y -80.5883,Z 121,A -139.9323,B 24.9544,C -1.5597,E1 24.8845,E2 225.9816} C_DIS
LIN {X -82.0192,Y -84.092,Z 121,A -137.4604,B 24.9545,C -1.5578,E1 24.8894,E2 223.5038} C_DIS
LIN {X -79.3648,Y -86.5989,Z 121,A -135.7582,B 24.9549,C -1.5508,E1 24.8929,E2 221.8113} C_DIS
LIN {X -76.776,Y -88.9045,Z 121,A -134.1143,B 24.9553,C -1.5454,E1 24.8963,E2 220.1737} C_DIS
LIN {X -73.5801,Y -91.5661,Z 121,A -131.9406,B 24.9551,C -1.5478,E1 24.901,E2 217.986} C_DIS
LIN {X -70.7046,Y -93.8031,Z 121,A -130.3748,B 24.9558,C -1.5355,E1 24.9044,E2 216.4438} C_DIS
LIN {X -68.7447,Y -95.2506,Z 121,A -128.9388,B 24.9553,C -1.5441,E1 24.9077,E2 214.9822} C_DIS
LIN {X -65.7672,Y -97.3284,Z 121,A -127.2548,B 24.9557,C -1.5375,E1 24.9116,E2 213.3084} C_DIS
LIN {X -62.7507,Y -99.3018,Z 121,A -125.4017,B 24.9557,C -1.5388,E1 24.916,E2 211.4462} C_DIS
LIN {X -60.0157,Y -100.9769,Z 121,A -123.952,B 24.9561,C -1.5315,E1 24.9194,E2 210.0094} C_DIS
LIN {X -57.3493,Y -102.5144,Z 121,A -122.337,B 24.9559,C -1.5344,E1 24.9234,E2 208.3829} C_DIS
LIN {X -53.8792,Y -104.381,Z 121,A -120.4191,B 24.956,C -1.5317,E1 24.9281,E2 206.4662} C_DIS
LIN {X -50.3124,Y -106.147,Z 121,A -118.4435,B 24.956,C -1.5308,E1 24.9331,E2 204.4874} C_DIS
LIN {X -47.009,Y -107.6489,Z 121,A -116.7275,B 24.9563,C -1.5265,E1 24.9374,E2 202.7777} C_DIS
LIN {X -43.1896,Y -109.2376,Z 121,A -114.75,B 24.9566,C -1.5226,E1 24.9425,E2 200.8048} C_DIS
LIN {X -40.4795,Y -110.2706,Z 121,A -112.0472,B 24.9533,C -1.5792,E1 24.9501,E2 197.9624} C_DIS
LIN {X -33.287,Y -112.6505,Z 121,A -109.9414,B 24.9576,C -1.5049,E1 24.9552,E2 196.0292} C_DIS
LIN {X -29.9898,Y -113.5746,Z 121,A -107.8447,B 24.9566,C -1.5228,E1 24.9609,E2 193.8868} C_DIS
LIN {X -26.3643,Y -114.4686,Z 121,A -106.1706,B 24.957,C -1.5153,E1 24.9654,E2 192.2283} C_DIS
LIN {X -23.0894,Y -115.1751,Z 121,A -104.4831,B 24.9569,C -1.5169,E1 24.9701,E2 190.5348} C_DIS
LIN {X -20.1568,Y -115.7249,Z 121,A -103.0811,B 24.9571,C -1.514,E1 24.9739,E2 189.1383} C_DIS
LIN {X -16.6179,Y -116.2841,Z 121,A -101.3363,B 24.9571,C -1.5135,E1 24.9787,E2 187.3934} C_DIS
LIN {X -13.4337,Y -116.695,Z 121,A -99.7072,B 24.9569,C -1.5161,E1 24.9833,E2 185.757} C_DIS
LIN {X -9.6354,Y -117.0699,Z 121,A -97.9044,B 24.9571,C -1.5133,E1 24.9883,E2 183.9599} C_DIS
LIN {X -6.2546,Y -117.299,Z 121,A -96.2283,B 24.9571,C -1.5144,E1 24.9929,E2 182.2806} C_DIS
LIN {X -2.1973,Y -117.4449,Z 121,A -94.2612,B 24.9571,C -1.5141,E1 24.9984,E2 180.3141} C_DIS
LIN {X 0.8321,Y -117.4596,Z 121,A -93.3379,B 24.9584,C -1.4893,E1 25.0009,E2 179.4494} C_DIS
Enddeposition()
LIN {X 0.8321,Y -117.4596,Z 121,A -93.3379,B 24.9584,C -1.4893,E1 25.0009,E2 179.4494} C_DIS
Startdeposition()
$VEL.CP = VEL_PRINT
LIN {X -0.7505,Y -116.5814,Z 121,A -94.3235,B 24.9581,C -1.4953,E1 24.9981,E2 180.4208} C_DIS
LIN {X -4.6276,Y -116.4925,Z 121,A -96.2469,B 24.9581,C -1.4943,E1 24.9928,E2 182.3469} C_DIS
LIN {X -7.9922,Y -116.3096,Z 121,A -97.8524,B 24.9581,C -1.4965,E1 24.9883,E2 183.9478} C_DIS
LIN {X -11.7385,Y -115.992,Z 121,A -99.7788,B 24.9582,C -1.4931,E1 24.9829,E2 185.8831} C_DIS
LIN {X -15.2044,Y -115.5883,Z 121,A -101.8987,B 24.9592,C -1.4756,E1 24.9769,E2 188.046} C_DIS
LIN {X -18.8915,Y -115.0435,Z 121,A -103.0568,B 24.9575,C -1.5057,E1 24.9739,E2 189.1338} C_DIS
LIN {X -22.3171,Y -114.4282,Z 121,A -104.9209,B 24.9579,C -1.4995,E1 24.9688,E2 191.0144} C_DIS
LIN {X -26.3066,Y -113.577,Z 121,A -107.0173,B 24.958,C -1.4965,E1 24.963,E2 193.1207} C_DIS
LIN {X -30.0671,Y -112.6404,Z 121,A -108.8173,B 24.9577,C -1.5022,E1 24.9582,E2 194.9098} C_DIS
LIN {X -32.3462,Y -112.0082,Z 121,A -110.3337,B 24.9585,C -1.4875,E1 24.954,E2 196.4634} C_DIS
LIN {X -39.2427,Y -109.7827,Z 121,A -113.5562,B 24.9576,C -1.5051,E1 24.9456,E2 199.6502} C_DIS
LIN {X -43.1846,Y -108.2923,Z 121,A -115.7486,B 24.9577,C -1.5018,E1 24.9398,E2 201.855} C_DIS
LIN {X -45.7266,Y -107.2431,Z 121,A -117.1315,B 24.9577,C -1.5019,E1 24.9362,E2 203.2409} C_DIS
LIN {X -49.2601,Y -105.6656,Z 121,A -118.9979,B 24.9575,C -1.5056,E1 24.9315,E2 205.1031} C_DIS
LIN {X -53.5205,Y -103.5742,Z 121,A -121.656,B 24.9581,C -1.4946,E1 24.9248,E2 207.7943} C_DIS
LIN {X -56.3643,Y -102.0546,Z 121,A -122.7707,B 24.9569,C -1.5168,E1 24.9222,E2 208.8595} C_DIS
LIN {X -60.7166,Y -99.5254,Z 121,A -125.3543,B 24.9569,C -1.5158,E1 24.916,E2 211.4534} C_DIS
LIN {X -63.4127,Y -97.8309,Z 121,A -126.8884,B 24.9567,C -1.5195,E1 24.9123,E2 212.9836} C_DIS
LIN {X -66.0638,Y -96.0609,Z 121,A -128.6236,B 24.957,C -1.5149,E1 24.9083,E2 214.7355} C_DIS
LIN {X -69.0757,Y -93.9169,Z 121,A -130.2763,B 24.9564,C -1.525,E1 24.9046,E2 216.3699} C_DIS
LIN {X -71.7274,Y -91.9101,Z 121,A -132.1326,B 24.9568,C -1.5186,E1 24.9004,E2 218.2484} C_DIS
LIN {X -76.9949,Y -87.5427,Z 121,A -135.2561,B 24.9558,C -1.5351,E1 24.8938,E2 221.3445} C_DIS
LIN {X -78.9834,Y -85.7522,Z 121,A -137.5513,B 24.958,C -1.497,E1 24.8889,E2 223.7398} C_DIS
LIN {X -82.9582,Y -81.9128,Z 121,A -139.0314,B 24.9547,C -1.5542,E1 24.8863,E2 225.0899} C_DIS
LIN {X -84.7756,Y -80.0308,Z 121,A -140.7022,B 24.9555,C -1.5409,E1 24.8829,E2 226.7997} C_DIS
LIN {X -87.0381,Y -77.5642,Z 121,A -142.8265,B 24.9564,C -1.5247,E1 24.8789,E2 228.9719} C_DIS
LIN {X -89.4914,Y -74.7204,Z 121,A -144.172,B 24.955,C -1.5497,E1 24.8766,E2 230.264} C_DIS
LIN {X -93.6779,Y -69.4022,Z 121,A -147.4789,B 24.9545,C -1.5586,E1 24.8709,E2 233.5655} C_DIS
LIN {X -95.5085,Y -66.8585,Z 121,A -149.4559,B 24.9553,C -1.5445,E1 24.8676,E2 235.5858} C_DIS
LIN {X -97.6404,Y -63.7059,Z 121,A -151.0502,B 24.9544,C -1.5606,E1 24.8652,E2 237.1495} C_DIS
LIN {X -99.6106,Y -60.5764,Z 121,A -152.8324,B 24.954,C -1.5669,E1 24.8626,E2 238.9259} C_DIS
LIN {X -101.2877,Y -57.73,Z 121,A -154.466,B 24.9538,C -1.5709,E1 24.8603,E2 240.5584} C_DIS
LIN {X -103.198,Y -54.2398,Z 121,A -156.409,B 24.9534,C -1.5768,E1 24.8578,E2 242.4976} C_DIS
LIN {X -104.6737,Y -51.3365,Z 121,A -158.237,B 24.9537,C -1.572,E1 24.8555,E2 244.347} C_DIS
LIN {X -106.4227,Y -47.6034,Z 121,A -160.5871,B 24.9541,C -1.5647,E1 24.8527,E2 246.7275} C_DIS
LIN {X -107.9812,Y -43.9527,Z 121,A -162.0297,B 24.9526,C -1.591,E1 24.8513,E2 248.1153} C_DIS
LIN {X -109.131,Y -41.0156,Z 121,A -163.5719,B 24.9523,C -1.5959,E1 24.8497,E2 249.6544} C_DIS
LIN {X -110.518,Y -37.1155,Z 121,A -165.574,B 24.9518,C -1.6034,E1 24.8479,E2 251.6502} C_DIS
LIN {X -111.4097,Y -34.3467,Z 121,A -167.0743,B 24.9518,C -1.6048,E1 24.8466,E2 253.1557} C_DIS
LIN {X -112.4876,Y -30.6329,Z 121,A -169.0339,B 24.9515,C -1.6083,E1 24.8451,E2 255.1184} C_DIS
LIN {X -113.4042,Y -27.0485,Z 121,A -170.9297,B 24.9514,C -1.6108,E1 24.8439,E2 257.0194} C_DIS
LIN {X -114.4687,Y -22.1063,Z 121,A -173.1616,B 24.9503,C -1.6288,E1 24.8426,E2 259.2213} C_DIS
LIN {X -115.1485,Y -18.2428,Z 121,A -175.6198,B 24.9512,C -1.6135,E1 24.8414,E2 261.7307} C_DIS
LIN {X -115.606,Y -15.0678,Z 121,A -176.8338,B 24.95,C -1.6332,E1 24.841,E2 262.905} C_DIS
LIN {X -116.0055,Y -11.6099,Z 121,A -179.1286,B 24.9511,C -1.6151,E1 24.8403,E2 265.2566} C_DIS
LIN {X -116.342,Y -7.5131,Z 121,A 178.9791,B 24.9504,C -1.6268,E1 24.84,E2 267.1325} C_DIS
LIN {X -116.5163,Y -3.9878,Z 121,A 177.678,B 24.949,C -1.6499,E1 24.8399,E2 268.3864} C_DIS
LIN {X -116.5818,Y -0.7584,Z 121,A 175.567,B 24.95,C -1.634,E1 24.8398,E2 270.548} C_DIS
LIN {X -116.544,Y 3.0853,Z 121,A 174.1306,B 24.9485,C -1.6583,E1 24.8398,E2 271.9351} C_DIS
LIN {X -116.291,Y 8.2665,Z 121,A 171.902,B 24.9471,C -1.6796,E1 24.8402,E2 274.1263} C_DIS
LIN {X -116.0795,Y 10.8321,Z 121,A 170.2638,B 24.9478,C -1.6686,E1 24.8406,E2 275.8005} C_DIS
LIN {X -115.653,Y 14.7046,Z 121,A 168.2209,B 24.9478,C -1.6697,E1 24.8413,E2 277.8531} C_DIS
LIN {X -114.8837,Y 19.8454,Z 121,A 165.8049,B 24.9469,C -1.6835,E1 24.8423,E2 280.2505} C_DIS
LIN {X -114.11,Y 23.8932,Z 121,A 162.675,B 24.9492,C -1.646,E1 24.8442,E2 283.4882} C_DIS
LIN {X -112.6027,Y 30.2067,Z 121,A 160.8334,B 24.9452,C -1.7102,E1 24.8454,E2 285.1876} C_DIS
LIN {X -111.8251,Y 32.9692,Z 121,A 159.0865,B 24.9458,C -1.701,E1 24.8467,E2 286.9665} C_DIS
LIN {X -110.1011,Y 38.3354,Z 121,A 156.4424,B 24.9449,C -1.7148,E1 24.849,E2 289.5928} C_DIS
LIN {X -109.0554,Y 41.2152,Z 121,A 154.8157,B 24.9449,C -1.7147,E1 24.8506,E2 291.2291} C_DIS
LIN {X -107.7731,Y 44.4638,Z 121,A 152.6073,B 24.9458,C -1.7001,E1 24.853,E2 293.4843} C_DIS
LIN {X -106.2755,Y 47.93,Z 121,A 150.5526,B 24.946,C -1.6979,E1 24.8554,E2 295.5557} C_DIS
LIN {X -104.2423,Y 52.2067,Z 121,A 148.9573,B 24.9436,C -1.7343,E1 24.8572,E2 297.0729} C_DIS
LIN {X -102.6887,Y 55.1996,Z 121,A 146.7163,B 24.9448,C -1.7156,E1 24.8602,E2 299.3702} C_DIS
LIN {X -100.7465,Y 58.6718,Z 121,A 145.321,B 24.943,C -1.7439,E1 24.8621,E2 300.7053} C_DIS
LIN {X -98.3183,Y 62.6533,Z 121,A 142.8909,B 24.943,C -1.7449,E1 24.8657,E2 303.1455} C_DIS
LIN {X -96.3991,Y 65.5672,Z 121,A 141.2264,B 24.9425,C -1.7518,E1 24.8682,E2 304.8019} C_DIS
LIN {X -93.1484,Y 70.1082,Z 121,A 138.3666,B 24.9423,C -1.7547,E1 24.873,E2 307.6687} C_DIS
LIN {X -90.8049,Y 73.1189,Z 121,A 136.5758,B 24.9417,C -1.7631,E1 24.876,E2 309.4479} C_DIS
LIN {X -88.5406,Y 75.8448,Z 121,A 134.8889,B 24.9413,C -1.7699,E1 24.8791,E2 311.1263} C_DIS
LIN {X -86.4085,Y 78.2676,Z 121,A 133.0966,B 24.9416,C -1.7655,E1 24.8824,E2 312.9371} C_DIS
LIN {X -83.8554,Y 80.9942,Z 121,A 131.3751,B 24.941,C -1.7748,E1 24.8857,E2 314.644} C_DIS
LIN {X -81.0824,Y 83.7704,Z 121,A 129.4054,B 24.9408,C -1.7778,E1 24.8896,E2 316.6149} C_DIS
LIN {X -78.5051,Y 86.1911,Z 121,A 127.6026,B 24.9407,C -1.7792,E1 24.8933,E2 318.4216} C_DIS
LIN {X -75.5794,Y 88.7667,Z 121,A 125.7776,B 24.9401,C -1.7873,E1 24.8972,E2 320.2345} C_DIS
LIN {X -72.5658,Y 91.2475,Z 121,A 123.7894,B 24.9401,C -1.7886,E1 24.9015,E2 322.2269} C_DIS
LIN {X -69.7481,Y 93.4189,Z 121,A 122.1266,B 24.9395,C -1.7959,E1 24.9052,E2 323.8785} C_DIS
LIN {X -64.8611,Y 96.8772,Z 121,A 119.1856,B 24.9391,C -1.8019,E1 24.9119,E2 326.8153} C_DIS
LIN {X -62.2821,Y 98.555,Z 121,A 117.5072,B 24.9394,C -1.7978,E1 24.9159,E2 328.5087} C_DIS
LIN {X -58.9239,Y 100.598,Z 121,A 115.6645,B 24.9389,C -1.8051,E1 24.9202,E2 330.3398} C_DIS
LIN {X -55.7233,Y 102.4047,Z 121,A 113.7118,B 24.9391,C -1.8022,E1 24.925,E2 332.305} C_DIS
LIN {X -52.3533,Y 104.1696,Z 121,A 111.8018,B 24.9391,C -1.8036,E1 24.9298,E2 334.2169} C_DIS
LIN {X -45.0307,Y 107.5364,Z 121,A 108.0352,B 24.9381,C -1.8177,E1 24.9393,E2 337.959} C_DIS
LIN {X -40.6289,Y 109.2775,Z 121,A 105.7315,B 24.9378,C -1.8218,E1 24.9453,E2 340.2579} C_DIS
LIN {X -37.8862,Y 110.2581,Z 121,A 104.2085,B 24.9379,C -1.8197,E1 24.9493,E2 341.7888} C_DIS
LIN {X -34.4009,Y 111.3929,Z 121,A 102.483,B 24.9376,C -1.8251,E1 24.9539,E2 343.5046} C_DIS
LIN {X -31.5385,Y 112.2371,Z 121,A 100.8968,B 24.9378,C -1.8216,E1 24.9582,E2 345.1017} C_DIS
LIN {X -24.3254,Y 114.019,Z 121,A 96.5455,B 24.9396,C -1.7954,E1 24.9702,E2 349.5209} C_DIS
LIN {X -19.3937,Y 114.9595,Z 121,A 95.13,B 24.9364,C -1.8421,E1 24.9738,E2 350.8271} C_DIS
LIN {X -16.0585,Y 115.473,Z 121,A 93.1143,B 24.9374,C -1.8278,E1 24.9795,E2 352.8783} C_DIS
LIN {X -10.7413,Y 116.0879,Z 121,A 90.4836,B 24.9373,C -1.8292,E1 24.9868,E2 355.5072} C_DIS
LIN {X -7.3182,Y 116.3551,Z 121,A 88.888,B 24.937,C -1.8339,E1 24.9912,E2 357.0924} C_DIS
LIN {X -4.399,Y 116.5023,Z 121,A 87.3067,B 24.9374,C -1.8281,E1 24.9956,E2 358.6877} C_DIS
LIN {X -0.3331,Y 116.5839,Z 121,A 85.3806,B 24.9371,C -1.8317,E1 25.001,E2 360.6053} C_DIS
LIN {X 3.9233,Y 116.5183,Z 121,A 83.2355,B 24.9372,C -1.8297,E1 25.007,E2 362.7549} C_DIS
LIN {X 7.776,Y 116.3242,Z 121,A 81.4013,B 24.9371,C -1.8324,E1 25.0121,E2 364.582} C_DIS
LIN {X 11.7536,Y 115.9904,Z 121,A 79.3743,B 24.9373,C -1.8293,E1 25.0177,E2 366.615} C_DIS
LIN {X 16.036,Y 115.4762,Z 121,A 77.552,B 24.9364,C -1.8419,E1 25.0227,E2 368.406} C_DIS
LIN {X 20.4301,Y 114.7799,Z 121,A 74.9079,B 24.9378,C -1.8211,E1 25.0301,E2 371.0968} C_DIS
LIN {X 24.0922,Y 114.0692,Z 121,A 73.1639,B 24.9376,C -1.8241,E1 25.0349,E2 372.8315} C_DIS
LIN {X 28.2834,Y 113.1029,Z 121,A 71.2688,B 24.937,C -1.8326,E1 25.0399,E2 374.7038} C_DIS
LIN {X 32.2273,Y 112.0419,Z 121,A 68.6721,B 24.9389,C -1.8052,E1 25.0471,E2 377.3611} C_DIS
LIN {X 36.1028,Y 110.8531,Z 121,A 67.207,B 24.9374,C -1.8269,E1 25.0509,E2 378.7721} C_DIS
LIN {X 39.8621,Y 109.5573,Z 121,A 65.284,B 24.9374,C -1.8266,E1 25.0559,E2 380.692} C_DIS
LIN {X 42.9055,Y 108.4019,Z 121,A 63.6321,B 24.9377,C -1.8226,E1 25.0602,E2 382.3496} C_DIS
LIN {X 46.5122,Y 106.9037,Z 121,A 61.7504,B 24.9377,C -1.8222,E1 25.065,E2 384.2278} C_DIS
LIN {X 50.2022,Y 105.2218,Z 121,A 60.0004,B 24.9372,C -1.8308,E1 25.0694,E2 385.953} C_DIS
LIN {X 53.745,Y 103.4586,Z 121,A 57.7873,B 24.9382,C -1.8161,E1 25.075,E2 388.1948} C_DIS
LIN {X 56.9458,Y 101.7299,Z 121,A 56.0463,B 24.9382,C -1.8158,E1 25.0793,E2 389.9316} C_DIS
LIN {X 60.3014,Y 99.7777,Z 121,A 54.1307,B 24.9384,C -1.8126,E1 25.0839,E2 391.8488} C_DIS
LIN {X 63.1874,Y 97.9754,Z 121,A 52.4254,B 24.9387,C -1.8085,E1 25.0879,E2 393.5585} C_DIS
LIN {X 66.5034,Y 95.7553,Z 121,A 50.5061,B 24.9387,C -1.8071,E1 25.0923,E2 395.4744} C_DIS
LIN {X 69.7518,Y 93.4161,Z 121,A 48.1852,B 24.9401,C -1.7876,E1 25.0976,E2 397.8333} C_DIS
LIN {X 72.4213,Y 91.3617,Z 121,A 46.569,B 24.9401,C -1.7863,E1 25.1012,E2 399.4465} C_DIS
LIN {X 75.0378,Y 89.2276,Z 121,A 45.3272,B 24.9391,C -1.8021,E1 25.1037,E2 400.6462} C_DIS
LIN {X 76.9749,Y 87.5602,Z 121,A 43.967,B 24.9396,C -1.7948,E1 25.1066,E2 402.0181} C_DIS
LIN {X 80.5601,Y 84.2738,Z 121,A 41.7673,B 24.9394,C -1.7986,E1 25.1111,E2 404.1998} C_DIS
LIN {X 82.857,Y 82.0153,Z 121,A 40.0788,B 24.9399,C -1.7904,E1 25.1145,E2 405.9007} C_DIS
LIN {X 86.3385,Y 78.3445,Z 121,A 37.4821,B 24.9406,C -1.7797,E1 25.1194,E2 408.5113} C_DIS
LIN {X 88.8058,Y 75.5335,Z 121,A 35.7123,B 24.9407,C -1.7786,E1 25.1226,E2 410.2758} C_DIS
LIN {X 91.5803,Y 72.1447,Z 121,A 33.6914,B 24.9407,C -1.7795,E1 25.1262,E2 412.2851} C_DIS
LIN {X 92.9875,Y 70.3224,Z 121,A 32.4335,B 24.9412,C -1.7708,E1 25.1283,E2 413.5575} C_DIS
LIN {X 95.6496,Y 66.6554,Z 121,A 29.7539,B 24.943,C -1.7442,E1 25.1327,E2 416.2867} C_DIS
LIN {X 97.9071,Y 63.2939,Z 121,A 28.4967,B 24.9411,C -1.7731,E1 25.1346,E2 417.4697} C_DIS
LIN {X 99.9233,Y 60.0618,Z 121,A 26.304,B 24.9424,C -1.7531,E1 25.1378,E2 419.6984} C_DIS
LIN {X 101.8243,Y 56.7768,Z 121,A 24.5768,B 24.9424,C -1.7545,E1 25.1402,E2 421.4134} C_DIS
LIN {X 103.7656,Y 53.1459,Z 121,A 22.1932,B 24.9438,C -1.732,E1 25.1433,E2 423.8373} C_DIS
LIN {X 105.2801,Y 50.0807,Z 121,A 21.1729,B 24.9421,C -1.7581,E1 25.1445,E2 424.7905} C_DIS
LIN {X 106.9051,Y 46.5088,Z 121,A 18.9639,B 24.9433,C -1.7394,E1 25.147,E2 427.0318} C_DIS
LIN {X 108.3621,Y 43.0069,Z 121,A 17.082,B 24.9437,C -1.733,E1 25.149,E2 428.9183} C_DIS
LIN {X 109.6127,Y 39.7102,Z 121,A 15.4414,B 24.9437,C -1.7322,E1 25.1506,E2 430.5517} C_DIS
LIN {X 110.7949,Y 36.2827,Z 121,A 12.5129,B 24.9475,C -1.6732,E1 25.1533,E2 433.6027} C_DIS
LIN {X 112.7183,Y 29.7788,Z 121,A 10.4245,B 24.9445,C -1.7211,E1 25.1547,E2 435.566} C_DIS
LIN {X 114.3872,Y 22.5297,Z 121,A 6.79,B 24.9452,C -1.7107,E1 25.157,E2 439.2041} C_DIS
LIN {X 115.0774,Y 18.6883,Z 121,A 4.8924,B 24.9455,C -1.7055,E1 25.1579,E2 441.1027} C_DIS
LIN {X 115.4689,Y 16.0878,Z 121,A 3.3886,B 24.9464,C -1.6914,E1 25.1585,E2 442.631} C_DIS
LIN {X 115.9467,Y 12.1713,Z 121,A 1.5648,B 24.9464,C -1.6906,E1 25.159,E2 444.4458} C_DIS
LIN {X 116.2432,Y 8.9122,Z 121,A 0.0269,B 24.9466,C -1.6888,E1 25.1594,E2 445.979} C_DIS
LIN {X 116.4596,Y 5.3944,Z 121,A -1.7934,B 24.9472,C -1.6789,E1 25.1597,E2 447.8116} C_DIS
LIN {X 116.5683,Y 1.9163,Z 121,A -3.3793,B 24.9472,C -1.6793,E1 25.1597,E2 449.3873} C_DIS
LIN {X 116.5745,Y -1.5755,Z 121,A -5.254,B 24.948,C -1.6661,E1 25.1597,E2 451.2818} C_DIS
LIN {X 116.4674,Y -5.2113,Z 121,A -6.8686,B 24.9478,C -1.6685,E1 25.1596,E2 452.8812} C_DIS
LIN {X 116.3016,Y -8.1101,Z 121,A -8.4182,B 24.9485,C -1.658,E1 25.1593,E2 454.4463} C_DIS
LIN {X 115.9605,Y -12.0395,Z 121,A -10.2662,B 24.9486,C -1.656,E1 25.1588,E2 456.2882} C_DIS
LIN {X 115.2684,Y -17.4672,Z 121,A -12.716,B 24.9484,C -1.6586,E1 25.1579,E2 458.7174} C_DIS
LIN {X 114.6263,Y -21.2841,Z 121,A -14.8698,B 24.9496,C -1.6404,E1 25.1569,E2 460.9014} C_DIS
LIN {X 113.9216,Y -24.7718,Z 121,A -16.5263,B 24.9496,C -1.6392,E1 25.1559,E2 462.5512} C_DIS
LIN {X 113.1914,Y -27.9208,Z 121,A -18.4055,B 24.9508,C -1.6202,E1 25.1547,E2 464.4642} C_DIS
LIN {X 112.0609,Y -32.1603,Z 121,A -20.4037,B 24.9508,C -1.6208,E1 25.1532,E2 466.4495} C_DIS
LIN {X 110.0917,Y -38.3621,Z 121,A -23.1951,B 24.9502,C -1.63,E1 25.1509,E2 469.2034} C_DIS
LIN {X 108.8862,Y -41.6621,Z 121,A -25.1702,B 24.9513,C -1.6128,E1 25.1489,E2 471.2082} C_DIS
LIN {X 107.1802,Y -45.8759,Z 121,A -27.4675,B 24.9519,C -1.6028,E1 25.1464,E2 473.5162} C_DIS
LIN {X 104.55,Y -51.5861,Z 121,A -30.4583,B 24.9521,C -1.5981,E1 25.1429,E2 476.502} C_DIS
LIN {X 103.1124,Y -54.4023,Z 121,A -31.9694,B 24.9523,C -1.5955,E1 25.1409,E2 478.0113} C_DIS
LIN {X 101.5176,Y -57.3259,Z 121,A -34.5311,B 24.9552,C -1.5472,E1 25.1373,E2 480.6737} C_DIS
LIN {X 98.5583,Y -62.2768,Z 121,A -36.3522,B 24.9528,C -1.5865,E1 25.1348,E2 482.3928} C_DIS
LIN {X 96.2383,Y -65.8047,Z 121,A -38.6218,B 24.9537,C -1.5714,E1 25.1312,E2 484.6867} C_DIS
LIN {X 94.0175,Y -68.9383,Z 121,A -40.3596,B 24.9537,C -1.5733,E1 25.1284,E2 486.4117} C_DIS
LIN {X 91.7665,Y -71.9091,Z 121,A -42.2668,B 24.9541,C -1.5647,E1 25.1251,E2 488.3301} C_DIS
LIN {X 89.5578,Y -74.6404,Z 121,A -43.9291,B 24.9542,C -1.5631,E1 25.1222,E2 489.9883} C_DIS
LIN {X 86.8435,Y -77.7816,Z 121,A -45.9309,B 24.9544,C -1.5596,E1 25.1185,E2 491.9895} C_DIS
LIN {X 84.4731,Y -80.3524,Z 121,A -48.3167,B 24.9565,C -1.5241,E1 25.1138,E2 494.4487} C_DIS
LIN {X 81.242,Y -83.6166,Z 121,A -50.5159,B 24.9566,C -1.5213,E1 25.1094,E2 496.6454} C_DIS
LIN {X 78.0213,Y -86.629,Z 121,A -51.846,B 24.9547,C -1.5552,E1 25.1068,E2 497.8901} C_DIS
LIN {X 75.8282,Y -88.5548,Z 121,A -53.8909,B 24.9565,C -1.5234,E1 25.1024,E2 500.002} C_DIS
LIN {X 73.1372,Y -90.7901,Z 121,A -55.4007,B 24.9562,C -1.5293,E1 25.0991,E2 501.4922} C_DIS
LIN {X 69.5216,Y -93.5891,Z 121,A -57.3844,B 24.9558,C -1.5367,E1 25.0948,E2 503.4513} C_DIS
LIN {X 66.7522,Y -95.5824,Z 121,A -59.1286,B 24.9561,C -1.5301,E1 25.0908,E2 505.205} C_DIS
LIN {X 63.6269,Y -97.6925,Z 121,A -61.0757,B 24.9566,C -1.522,E1 25.0862,E2 507.1647} C_DIS
LIN {X 60.417,Y -99.7075,Z 121,A -62.7532,B 24.9563,C -1.527,E1 25.0823,E2 508.825} C_DIS
LIN {X 57.8914,Y -101.1949,Z 121,A -64.23,B 24.9566,C -1.5227,E1 25.0787,E2 510.3076} C_DIS
LIN {X 52.2931,Y -104.1995,Z 121,A -67.2375,B 24.9566,C -1.5226,E1 25.0713,E2 513.3068} C_DIS
LIN {X 48.9111,Y -105.828,Z 121,A -69.1979,B 24.957,C -1.5143,E1 25.0663,E2 515.2817} C_DIS
LIN {X 45.3322,Y -107.4094,Z 121,A -71.5744,B 24.9584,C -1.4907,E1 25.0601,E2 517.7084} C_DIS
LIN {X 41.769,Y -108.8457,Z 121,A -72.8473,B 24.9569,C -1.5161,E1 25.0569,E2 518.9183} C_DIS
LIN {X 37.839,Y -110.2741,Z 121,A -75.1329,B 24.9577,C -1.5028,E1 25.0508,E2 521.2306} C_DIS
LIN {X 33.8349,Y -111.5683,Z 121,A -78.3331,B 24.9606,C -1.4495,E1 25.042,E2 524.5514} C_DIS
LIN {X 26.8808,Y -113.4444,Z 121,A -81.2321,B 24.9593,C -1.4745,E1 25.0343,E2 527.387} C_DIS
LIN {X 22.7468,Y -114.3426,Z 121,A -83.0822,B 24.9588,C -1.483,E1 25.0293,E2 529.2148} C_DIS
LIN {X 19.409,Y -114.957,Z 121,A -84.5986,B 24.9585,C -1.4885,E1 25.0251,E2 530.7165} C_DIS
LIN {X 16.1506,Y -115.4599,Z 121,A -86.0771,B 24.9582,C -1.4937,E1 25.0211,E2 532.1814} C_DIS
LIN {X 12.2034,Y -115.9433,Z 121,A -87.9787,B 24.9582,C -1.4949,E1 25.0158,E2 534.0787} C_DIS
LIN {X 7.9833,Y -116.3102,Z 121,A -90.0068,B 24.9581,C -1.4963,E1 25.0102,E2 536.1026} C_DIS
LIN {X 4.7452,Y -116.4875,Z 121,A -91.6789,B 24.9583,C -1.4922,E1 25.0055,E2 537.7838} C_DIS
LIN {X 0.8317,Y -116.5806,Z 121,A -93.5134,B 24.9581,C -1.4956,E1 25.0004,E2 539.6099} C_DIS
Enddeposition()
LIN {X 0.8317,Y -116.5806,Z 121,A -93.5134,B 24.9581,C -1.4956,E1 25.0004,E2 539.6099} C_DIS
Startdeposition()
$VEL.CP = VEL_PRINT
LIN {X 1.8015,Y -115.6885,Z 121,A -92.3174,B 24.9554,C -1.5432,E1 25.0041,E2 538.3015} C_DIS
LIN {X 5.2441,Y -115.5835,Z 121,A -90.7024,B 24.9556,C -1.5397,E1 25.0085,E2 536.695} C_DIS
LIN {X 8.665,Y -115.3785,Z 121,A -88.7099,B 24.9548,C -1.5538,E1 25.0142,E2 534.6701} C_DIS
LIN {X 13.2255,Y -114.944,Z 121,A -86.6577,B 24.9553,C -1.5453,E1 25.0198,E2 532.6393} C_DIS
LIN {X 16.264,Y -114.5533,Z 121,A -84.5898,B 24.9537,C -1.5714,E1 25.0257,E2 530.5114} C_DIS
LIN {X 20.4509,Y -113.8804,Z 121,A -82.6741,B 24.9541,C -1.5647,E1 25.0309,E2 528.6139} C_DIS
LIN {X 23.8699,Y -113.2139,Z 121,A -81.1042,B 24.9545,C -1.5591,E1 25.0352,E2 527.0591} C_DIS
LIN {X 28.3655,Y -112.1721,Z 121,A -78.1879,B 24.9526,C -1.5905,E1 25.0433,E2 524.0728} C_DIS
LIN {X 33.7708,Y -110.6651,Z 121,A -76.1598,B 24.9545,C -1.559,E1 25.0485,E2 522.1228} C_DIS
LIN {X 36.8177,Y -109.688,Z 121,A -74.6926,B 24.9547,C -1.5556,E1 25.0523,E2 520.6664} C_DIS
LIN {X 40.1175,Y -108.5256,Z 121,A -72.8806,B 24.9543,C -1.5615,E1 25.0571,E2 518.8442} C_DIS
LIN {X 47.175,Y -105.6487,Z 121,A -69.4182,B 24.9548,C -1.5526,E1 25.066,E2 515.4108} C_DIS
LIN {X 50.4829,Y -104.1087,Z 121,A -66.3124,B 24.9511,C -1.6162,E1 25.0742,E2 512.1631} C_DIS
LIN {X 56.3522,Y -101.0515,Z 121,A -64.4983,B 24.9548,C -1.5535,E1 25.0782,E2 510.5023} C_DIS
LIN {X 59.9104,Y -98.9837,Z 121,A -62.0625,B 24.9535,C -1.5757,E1 25.0842,E2 508.0214} C_DIS
LIN {X 63.1403,Y -96.9573,Z 121,A -60.1286,B 24.9531,C -1.5815,E1 25.0887,E2 506.0801} C_DIS
LIN {X 66.055,Y -94.9932,Z 121,A -58.5412,B 24.9534,C -1.5779,E1 25.0924,E2 504.5066} C_DIS
LIN {X 68.6868,Y -93.1089,Z 121,A -56.9625,B 24.9532,C -1.5801,E1 25.0959,E2 502.9282} C_DIS
LIN {X 74.3707,Y -88.6356,Z 121,A -53.3175,B 24.9526,C -1.5909,E1 25.1039,E2 499.2713} C_DIS
LIN {X 77.1406,Y -86.234,Z 121,A -51.5426,B 24.9524,C -1.5933,E1 25.1076,E2 497.4979} C_DIS
LIN {X 80.9478,Y -82.6722,Z 121,A -48.5601,B 24.9509,C -1.6185,E1 25.1137,E2 494.4683} C_DIS
LIN {X 83.3867,Y -80.21,Z 121,A -47.2899,B 24.9519,C -1.6016,E1 25.1161,E2 493.2433} C_DIS
LIN {X 85.6093,Y -77.8351,Z 121,A -45.4386,B 24.951,C -1.6171,E1 25.1197,E2 491.3637} C_DIS
LIN {X 87.7887,Y -75.3679,Z 121,A -43.9586,B 24.9512,C -1.6143,E1 25.1223,E2 489.8971} C_DIS
LIN {X 90.3085,Y -72.3311,Z 121,A -41.998,B 24.9508,C -1.6198,E1 25.1258,E2 487.9325} C_DIS
LIN {X 92.656,Y -69.2957,Z 121,A -40.2236,B 24.9508,C -1.619,E1 25.1288,E2 486.1683} C_DIS
LIN {X 94.8883,Y -66.2059,Z 121,A -38.3328,B 24.9506,C -1.6244,E1 25.1319,E2 484.274} C_DIS
LIN {X 96.7424,Y -63.4661,Z 121,A -36.717,B 24.9503,C -1.628,E1 25.1344,E2 482.6578} C_DIS
LIN {X 100.2641,Y -57.7417,Z 121,A -32.7471,B 24.9478,C -1.6684,E1 25.1401,E2 478.613} C_DIS
LIN {X 102.4884,Y -53.6952,Z 121,A -29.9439,B 24.9458,C -1.7003,E1 25.1438,E2 475.7495} C_DIS
LIN {X 105.544,Y -47.4073,Z 121,A -27.8126,B 24.9492,C -1.6467,E1 25.1462,E2 473.756} C_DIS
LIN {X 107.2218,Y -43.4796,Z 121,A -25.5737,B 24.9484,C -1.6592,E1 25.1486,E2 471.5} C_DIS
LIN {X 108.5883,Y -39.9456,Z 121,A -23.6908,B 24.948,C -1.6653,E1 25.1504,E2 469.613} C_DIS
LIN {X 110.5625,Y -34.1019,Z 121,A -20.7521,B 24.9478,C -1.6695,E1 25.153,E2 466.6812} C_DIS
LIN {X 111.3974,Y -31.2678,Z 121,A -19.1509,B 24.9471,C -1.6807,E1 25.1543,E2 465.0627} C_DIS
LIN {X 112.5602,Y -26.7881,Z 121,A -16.8154,B 24.9465,C -1.6902,E1 25.1558,E2 462.7184} C_DIS
LIN {X 113.2984,Y -23.4625,Z 121,A -15.2503,B 24.9465,C -1.6898,E1 25.1567,E2 461.1633} C_DIS
LIN {X 113.9382,Y -20.1295,Z 121,A -13.6559,B 24.9465,C -1.6911,E1 25.1575,E2 459.5751} C_DIS
LIN {X 114.9388,Y -13.2698,Z 121,A -10.3889,B 24.9462,C -1.6944,E1 25.1588,E2 456.3198} C_DIS
LIN {X 115.2205,Y -10.5459,Z 121,A -8.8417,B 24.9453,C -1.7079,E1 25.1592,E2 454.7497} C_DIS
LIN {X 115.513,Y -6.6167,Z 121,A -6.8903,B 24.9449,C -1.7143,E1 25.1596,E2 452.7949} C_DIS
LIN {X 115.6628,Y -3.0544,Z 121,A -5.0852,B 24.9444,C -1.7219,E1 25.1598,E2 450.9825} C_DIS
LIN {X 115.6983,Y 1.0214,Z 121,A -3.1979,B 24.9444,C -1.7223,E1 25.1598,E2 449.1057} C_DIS
LIN {X 115.6201,Y 4.3927,Z 121,A -1.4281,B 24.9438,C -1.7325,E1 25.1596,E2 447.3223} C_DIS
LIN {X 115.4203,Y 8.0742,Z 121,A 0.3802,B 24.9434,C -1.7376,E1 25.1593,E2 445.5127} C_DIS
LIN {X 115.062,Y 12.154,Z 121,A 2.3482,B 24.9432,C -1.7412,E1 25.1588,E2 443.5477} C_DIS
LIN {X 114.604,Y 15.9067,Z 121,A 4.2382,B 24.9427,C -1.7481,E1 25.1581,E2 441.6528} C_DIS
LIN {X 113.7216,Y 21.3233,Z 121,A 6.7608,B 24.9427,C -1.7474,E1 25.1569,E2 439.1465} C_DIS
LIN {X 112.6501,Y 26.4016,Z 121,A 9.3669,B 24.9421,C -1.7571,E1 25.1554,E2 436.5327} C_DIS
LIN {X 111.9233,Y 29.3333,Z 121,A 11.994,B 24.9382,C -1.816,E1 25.1534,E2 433.782} C_DIS
LIN {X 110.1138,Y 35.5236,Z 121,A 14.0751,B 24.9411,C -1.7724,E1 25.1518,E2 431.8155} C_DIS
LIN {X 109.1135,Y 38.4872,Z 121,A 15.6197,B 24.9408,C -1.7769,E1 25.1503,E2 430.269} C_DIS
LIN {X 107.9562,Y 41.6284,Z 121,A 17.4264,B 24.94,C -1.7888,E1 25.1485,E2 428.4442} C_DIS
LIN {X 106.507,Y 45.2031,Z 121,A 19.1987,B 24.94,C -1.7879,E1 25.1466,E2 426.6837} C_DIS
LIN {X 104.7046,Y 49.2353,Z 121,A 21.5451,B 24.9392,C -1.8017,E1 25.1439,E2 424.3175} C_DIS
LIN {X 102.2466,Y 54.1543,Z 121,A 23.9905,B 24.9395,C -1.7963,E1 25.1408,E2 421.898} C_DIS
LIN {X 100.7456,Y 56.9,Z 121,A 25.6998,B 24.9387,C -1.808,E1 25.1385,E2 420.1698} C_DIS
LIN {X 98.8833,Y 60.0755,Z 121,A 27.3836,B 24.9388,C -1.8064,E1 25.1361,E2 418.4985} C_DIS
LIN {X 97.2148,Y 62.7403,Z 121,A 29.7146,B 24.9361,C -1.847,E1 25.1324,E2 416.0833} C_DIS
LIN {X 94.3796,Y 66.9296,Z 121,A 31.4661,B 24.9381,C -1.8179,E1 25.1297,E2 414.4092} C_DIS
LIN {X 92.3595,Y 69.6905,Z 121,A 33.1256,B 24.9379,C -1.8205,E1 25.127,E2 412.7515} C_DIS
LIN {X 89.3611,Y 73.4977,Z 121,A 35.4141,B 24.9379,C -1.8211,E1 25.123,E2 410.4723} C_DIS
LIN {X 87.7653,Y 75.3953,Z 121,A 36.8189,B 24.9371,C -1.8322,E1 25.1204,E2 409.0476} C_DIS
LIN {X 83.259,Y 80.3425,Z 121,A 39.9714,B 24.9371,C -1.8322,E1 25.1145,E2 405.9091} C_DIS
LIN {X 81.0455,Y 82.5756,Z 121,A 41.7037,B 24.9363,C -1.8436,E1 25.111,E2 404.157} C_DIS
LIN {X 76.603,Y 86.7144,Z 121,A 44.6394,B 24.9361,C -1.8464,E1 25.105,E2 401.2266} C_DIS
LIN {X 73.6028,Y 89.2723,Z 121,A 47.266,B 24.9336,C -1.8815,E1 25.0992,E2 398.5272} C_DIS
LIN {X 69.6971,Y 92.3545,Z 121,A 48.7292,B 24.9366,C -1.8398,E1 25.0962,E2 397.1679} C_DIS
LIN {X 66.3272,Y 94.804,Z 121,A 51.0881,B 24.9354,C -1.8569,E1 25.0907,E2 394.7768} C_DIS
LIN {X 63.2124,Y 96.9097,Z 121,A 53.0255,B 24.9349,C -1.8634,E1 25.0862,E2 392.8305} C_DIS
LIN {X 60.0755,Y 98.8833,Z 121,A 54.7123,B 24.9352,C -1.8594,E1 25.0822,E2 391.1584} C_DIS
LIN {X 57.1638,Y 100.5961,Z 121,A 56.5082,B 24.9346,C -1.8674,E1 25.0778,E2 389.3489} C_DIS
LIN {X 53.8707,Y 102.3959,Z 121,A 58.2675,B 24.9348,C -1.8655,E1 25.0735,E2 387.5992} C_DIS
LIN {X 50.0116,Y 104.3352,Z 121,A 60.5172,B 24.9342,C -1.8732,E1 25.0679,E2 385.3373} C_DIS
LIN {X 46.1291,Y 106.1089,Z 121,A 62.4891,B 24.9345,C -1.8692,E1 25.0629,E2 383.3796} C_DIS
LIN {X 42.5974,Y 107.5757,Z 121,A 64.412,B 24.9343,C -1.8725,E1 25.0579,E2 381.4535} C_DIS
LIN {X 39.6631,Y 108.6914,Z 121,A 65.9267,B 24.9343,C -1.8722,E1 25.0539,E2 379.9427} C_DIS
LIN {X 36.6377,Y 109.7487,Z 121,A 67.5076,B 24.9343,C -1.8733,E1 25.0498,E2 378.3622} C_DIS
LIN {X 30.2589,Y 111.6753,Z 121,A 70.7912,B 24.9341,C -1.8749,E1 25.041,E2 375.0804} C_DIS
LIN {X 27.2187,Y 112.4551,Z 121,A 72.9054,B 24.9323,C -1.9008,E1 25.0351,E2 372.9078} C_DIS
LIN {X 23.2354,Y 113.345,Z 121,A 74.9563,B 24.9321,C -1.9031,E1 25.0295,E2 370.8542} C_DIS
LIN {X 19.0738,Y 114.1191,Z 121,A 76.0994,B 24.935,C -1.8616,E1 25.0266,E2 369.8107} C_DIS
LIN {X 12.906,Y 114.9814,Z 121,A 79.8733,B 24.9328,C -1.8927,E1 25.016,E2 365.9663} C_DIS
LIN {X 7.6711,Y 115.4476,Z 121,A 82.1088,B 24.934,C -1.8767,E1 25.0098,E2 363.7698} C_DIS
LIN {X 4.5096,Y 115.6151,Z 121,A 84.1751,B 24.9324,C -1.8985,E1 25.0039,E2 361.6524} C_DIS
LIN {X 0.9046,Y 115.6987,Z 121,A 85.258,B 24.9346,C -1.8674,E1 25.0011,E2 360.6432} C_DIS
LIN {X -3.6367,Y 115.645,Z 121,A 87.3528,B 24.9351,C -1.8602,E1 24.9953,E2 358.5656} C_DIS
LIN {X -6.1468,Y 115.5389,Z 121,A 89.0686,B 24.9337,C -1.8802,E1 24.9904,E2 356.802} C_DIS
LIN {X -11.5143,Y 115.1289,Z 121,A 91.8119,B 24.9336,C -1.8822,E1 24.9827,E2 354.0524} C_DIS
LIN {X -16.7678,Y 114.4817,Z 121,A 94.2924,B 24.9341,C -1.8745,E1 24.9759,E2 351.5884} C_DIS
LIN {X -21.0641,Y 113.7692,Z 121,A 96.7587,B 24.9333,C -1.8863,E1 24.969,E2 349.0917} C_DIS
LIN {X -25.2989,Y 112.903,Z 121,A 99.1339,B 24.9327,C -1.8945,E1 24.9625,E2 346.694} C_DIS
LIN {X -29.1911,Y 111.9599,Z 121,A 100.5359,B 24.9346,C -1.8675,E1 24.9589,E2 345.354} C_DIS
LIN {X -31.9488,Y 111.2044,Z 121,A 102.0493,B 24.9344,C -1.8702,E1 24.9548,E2 343.8319} C_DIS
LIN {X -35.3859,Y 110.1584,Z 121,A 103.8338,B 24.9346,C -1.8683,E1 24.95,E2 342.0487} C_DIS
LIN {X -38.4802,Y 109.1159,Z 121,A 105.3863,B 24.9349,C -1.8636,E1 24.946,E2 340.5045} C_DIS
LIN {X -44.4164,Y 106.8385,Z 121,A 108.4567,B 24.9354,C -1.8559,E1 24.938,E2 337.4457} C_DIS
LIN {X -47.63,Y 105.4437,Z 121,A 110.777,B 24.9339,C -1.8781,E1 24.932,E2 335.067} C_DIS
LIN {X -51.0139,Y 103.8495,Z 121,A 111.9906,B 24.936,C -1.8481,E1 24.9291,E2 333.9215} C_DIS
LIN {X -53.599,Y 102.539,Z 121,A 113.8575,B 24.9349,C -1.8639,E1 24.9243,E2 332.012} C_DIS
LIN {X -58.4621,Y 99.8468,Z 121,A 116.2221,B 24.9363,C -1.8427,E1 24.9187,E2 329.6909} C_DIS
LIN {X -61.7649,Y 97.8385,Z 121,A 118.3864,B 24.9359,C -1.8496,E1 24.9135,E2 327.5036} C_DIS
LIN {X -68.6262,Y 93.1532,Z 121,A 122.2702,B 24.9371,C -1.8316,E1 24.9047,E2 323.6493} C_DIS
LIN {X -70.6016,Y 91.6646,Z 121,A 123.692,B 24.9367,C -1.8372,E1 24.9014,E2 322.2091} C_DIS
LIN {X -73.5615,Y 89.308,Z 121,A 125.6224,B 24.9369,C -1.8354,E1 24.8972,E2 320.2757} C_DIS
LIN {X -76.2867,Y 86.9906,Z 121,A 127.3895,B 24.9371,C -1.8312,E1 24.8935,E2 318.5117} C_DIS
LIN {X -79.156,Y 84.3879,Z 121,A 129.2553,B 24.9376,C -1.8245,E1 24.8897,E2 316.6543} C_DIS
LIN {X -81.5689,Y 82.0586,Z 121,A 130.8973,B 24.9379,C -1.8197,E1 24.8864,E2 315.0168} C_DIS
LIN {X -84.1238,Y 79.4369,Z 121,A 132.7538,B 24.9381,C -1.817,E1 24.8828,E2 313.1587} C_DIS
LIN {X -86.3771,Y 76.9807,Z 121,A 134.3873,B 24.9384,C -1.8121,E1 24.8798,E2 311.5296} C_DIS
LIN {X -88.6237,Y 74.385,Z 121,A 136.217,B 24.9384,C -1.813,E1 24.8765,E2 309.6895} C_DIS
LIN {X -90.7592,Y 71.7617,Z 121,A 138.1647,B 24.9379,C -1.8198,E1 24.873,E2 307.7165} C_DIS
LIN {X -92.7819,Y 69.1281,Z 121,A 140.3974,B 24.9366,C -1.8397,E1 24.8693,E2 305.4255} C_DIS
LIN {X -96.1623,Y 64.3444,Z 121,A 142.3045,B 24.9399,C -1.7905,E1 24.8664,E2 303.6262} C_DIS
LIN {X -97.7152,Y 61.9607,Z 121,A 145.0122,B 24.9365,C -1.8401,E1 24.8622,E2 300.7864} C_DIS
LIN {X -101.3083,Y 55.8924,Z 121,A 147.2373,B 24.9408,C -1.7775,E1 24.8593,E2 298.6989} C_DIS
LIN {X -102.6243,Y 53.4371,Z 121,A 148.805,B 24.9405,C -1.7811,E1 24.8573,E2 297.1143} C_DIS
LIN {X -105.1558,Y 48.266,Z 121,A 151.4975,B 24.9415,C -1.766,E1 24.8541,E2 294.4433} C_DIS
LIN {X -106.6512,Y 44.8609,Z 121,A 153.4781,B 24.9415,C -1.766,E1 24.8518,E2 292.4516} C_DIS
LIN {X -108.1164,Y 41.2052,Z 121,A 155.3816,B 24.9421,C -1.7581,E1 24.8499,E2 290.5565} C_DIS
LIN {X -110.5066,Y 34.2821,Z 121,A 158.982,B 24.9429,C -1.7455,E1 24.8467,E2 286.9655} C_DIS
LIN {X -111.4549,Y 31.0649,Z 121,A 160.6659,B 24.9432,C -1.7411,E1 24.8454,E2 285.2823} C_DIS
LIN {X -113.2804,Y 23.5499,Z 121,A 164.4292,B 24.9442,C -1.7261,E1 24.843,E2 281.5329} C_DIS
LIN {X -113.8765,Y 20.4724,Z 121,A 166.11,B 24.9442,C -1.7262,E1 24.8421,E2 279.8417} C_DIS
LIN {X -114.6071,Y 15.8854,Z 121,A 168.7492,B 24.9437,C -1.7326,E1 24.841,E2 277.1717} C_DIS
LIN {X -115.1214,Y 11.5863,Z 121,A 170.7167,B 24.9447,C -1.7184,E1 24.8404,E2 275.2263} C_DIS
LIN {X -115.6245,Y 4.2913,Z 121,A 174.1856,B 24.9458,C -1.7003,E1 24.8399,E2 271.7795} C_DIS
LIN {X -115.6775,Y -2.3987,Z 121,A 177.0934,B 24.9475,C -1.6731,E1 24.8399,E2 268.9191} C_DIS
LIN {X -115.4,Y -8.3748,Z 121,A -178.6473,B 24.9448,C -1.7163,E1 24.8405,E2 264.5311} C_DIS
LIN {X -114.9236,Y -13.3997,Z 121,A -177.1661,B 24.948,C -1.6666,E1 24.8409,E2 263.1596} C_DIS
LIN {X -113.8857,Y -20.4211,Z 121,A -173.7175,B 24.9488,C -1.6526,E1 24.8424,E2 259.7239} C_DIS
LIN {X -113.1956,Y -23.9631,Z 121,A -171.625,B 24.9484,C -1.6593,E1 24.8435,E2 257.603} C_DIS
LIN {X -112.4092,Y -27.407,Z 121,A -169.7991,B 24.9485,C -1.657,E1 24.8447,E2 255.7719} C_DIS
LIN {X -111.4211,Y -31.1843,Z 121,A -167.8115,B 24.9488,C -1.6533,E1 24.8461,E2 253.7816} C_DIS
LIN {X -110.4671,Y -34.4095,Z 121,A -166.1861,B 24.9492,C -1.6465,E1 24.8474,E2 252.1629} C_DIS
LIN {X -109.4235,Y -37.6021,Z 121,A -164.2768,B 24.9489,C -1.6516,E1 24.8492,E2 250.2306} C_DIS
LIN {X -108.0734,Y -41.3188,Z 121,A -162.505,B 24.9497,C -1.6381,E1 24.8509,E2 248.4809} C_DIS
LIN {X -106.2814,Y -45.7311,Z 121,A -159.9758,B 24.9497,C -1.6383,E1 24.8536,E2 245.9373} C_DIS
LIN {X -103.972,Y -50.7669,Z 121,A -157.2418,B 24.9502,C -1.63,E1 24.8569,E2 243.2081} C_DIS
LIN {X -102.048,Y -54.5314,Z 121,A -155.2188,B 24.9507,C -1.6213,E1 24.8595,E2 241.1952} C_DIS
LIN {X -100.3164,Y -57.6506,Z 121,A -153.5297,B 24.9512,C -1.6133,E1 24.8618,E2 239.5163} C_DIS
LIN {X -98.49,Y -60.7218,Z 121,A -151.6555,B 24.9512,C -1.6129,E1 24.8645,E2 237.6334} C_DIS
LIN {X -95.0402,Y -65.9874,Z 121,A -148.7506,B 24.9523,C -1.596,E1 24.869,E2 234.7542} C_DIS
LIN {X -93.3259,Y -68.3904,Z 121,A -147.1618,B 24.9522,C -1.5976,E1 24.8716,E2 233.1539} C_DIS
LIN {X -89.4487,Y -73.392,Z 121,A -144.0175,B 24.9526,C -1.5904,E1 24.877,E2 230.012} C_DIS
LIN {X -86.1819,Y -77.1988,Z 121,A -141.7251,B 24.9534,C -1.5766,E1 24.8812,E2 227.7419} C_DIS
LIN {X -84.2969,Y -79.2528,Z 121,A -140.0895,B 24.953,C -1.5842,E1 24.8843,E2 226.081} C_DIS
LIN {X -81.9492,Y -81.6797,Z 121,A -137.5375,B 24.9509,C -1.618,E1 24.8895,E2 223.4379} C_DIS
LIN {X -77.9095,Y -85.541,Z 121,A -135.7074,B 24.9537,C -1.5724,E1 24.8931,E2 221.7088} C_DIS
LIN {X -73.1734,Y -89.6259,Z 121,A -132.7206,B 24.9543,C -1.5617,E1 24.8994,E2 218.736} C_DIS
LIN {X -70.3279,Y -91.8754,Z 121,A -130.6195,B 24.9537,C -1.5713,E1 24.9041,E2 216.6041} C_DIS
LIN {X -67.0336,Y -94.3054,Z 121,A -128.7775,B 24.9544,C -1.56,E1 24.9082,E2 214.7828} C_DIS
LIN {X -64.4304,Y -96.104,Z 121,A -127.0005,B 24.954,C -1.5663,E1 24.9123,E2 212.9847} C_DIS
LIN {X -61.0755,Y -98.2691,Z 121,A -124.615,B 24.9532,C -1.5809,E1 24.9181,E2 210.5571} C_DIS
LIN {X -57.6612,Y -100.3103,Z 121,A -123.5289,B 24.9556,C -1.54,E1 24.9205,E2 209.5648} C_DIS
LIN {X -55.3729,Y -101.5917,Z 121,A -121.6116,B 24.9541,C -1.5648,E1 24.9253,E2 207.5832} C_DIS
LIN {X -52.2153,Y -103.251,Z 121,A -119.8694,B 24.9543,C -1.5615,E1 24.9297,E2 205.8441} C_DIS
LIN {X -48.8185,Y -104.8986,Z 121,A -118.2177,B 24.955,C -1.5498,E1 24.9338,E2 204.2159} C_DIS
LIN {X -45.7105,Y -106.2913,Z 121,A -116.3524,B 24.9547,C -1.5557,E1 24.9386,E2 202.3322} C_DIS
LIN {X -42.3186,Y -107.6852,Z 121,A -114.77,B 24.9553,C -1.5438,E1 24.9426,E2 200.7747} C_DIS
LIN {X -39.4153,Y -108.7818,Z 121,A -113.1798,B 24.9553,C -1.5447,E1 24.9468,E2 199.1791} C_DIS
LIN {X -33.2176,Y -110.8317,Z 121,A -110.1243,B 24.9559,C -1.5344,E1 24.9549,E2 196.1425} C_DIS
LIN {X -30.2424,Y -111.6798,Z 121,A -108.0574,B 24.9546,C -1.5568,E1 24.9606,E2 194.019} C_DIS
LIN {X -26.6037,Y -112.6035,Z 121,A -106.0023,B 24.9541,C -1.5645,E1 24.9662,E2 191.943} C_DIS
LIN {X -22.6684,Y -113.4614,Z 121,A -104.5983,B 24.9557,C -1.5375,E1 24.9699,E2 190.6015} C_DIS
LIN {X -19.3988,Y -114.0647,Z 121,A -102.0354,B 24.9534,C -1.5778,E1 24.9772,E2 187.9405} C_DIS
LIN {X -13.9678,Y -114.857,Z 121,A -100.3089,B 24.956,C -1.533,E1 24.9817,E2 186.3191} C_DIS
LIN {X -11.3046,Y -115.1505,Z 121,A -98.7056,B 24.9553,C -1.5451,E1 24.9862,E2 184.686} C_DIS
LIN {X -7.4102,Y -115.4652,Z 121,A -96.936,B 24.9557,C -1.5377,E1 24.9911,E2 182.9332} C_DIS
LIN {X -3.6343,Y -115.645,Z 121,A -94.9831,B 24.9555,C -1.5416,E1 24.9966,E2 180.9708} C_DIS
LIN {X -0.107,Y -115.7036,Z 121,A -93.2014,B 24.9554,C -1.5434,E1 25.0016,E2 179.1847} C_DIS
LIN {X -0.107,Y -115.7036,Z 121,A -93.2014,B 24.9554,C -1.5434,E1 25.0016,E2 179.1847} C_DIS
Enddeposition()
LIN {X 0.8211,Y -114.8151,Z 121,A -93.3866,B 24.9561,C -1.5303,E1 25.001,E2 179.4009} C_DIS
Startdeposition()
$VEL.CP = VEL_PRINT
LIN {X -2.2629,Y -114.7982,Z 121,A -95.139,B 24.9567,C -1.5207,E1 24.996,E2 181.1763} C_DIS
LIN {X -6.1231,Y -114.6572,Z 121,A -97.0748,B 24.9567,C -1.5201,E1 24.9906,E2 183.1138} C_DIS
LIN {X -9.5626,Y -114.4223,Z 121,A -98.8879,B 24.9569,C -1.5161,E1 24.9855,E2 184.9371} C_DIS
LIN {X -12.4692,Y -114.1425,Z 121,A -100.2179,B 24.9566,C -1.5218,E1 24.9819,E2 186.2545} C_DIS
LIN {X -16.2939,Y -113.6585,Z 121,A -102.5567,B 24.9576,C -1.5043,E1 24.9753,E2 188.6366} C_DIS
LIN {X -19.7128,Y -113.1173,Z 121,A -103.947,B 24.9568,C -1.5193,E1 24.9716,E2 189.9926} C_DIS
LIN {X -24.0264,Y -112.2794,Z 121,A -106.1049,B 24.9566,C -1.5217,E1 24.9657,E2 192.1473} C_DIS
LIN {X -28.9991,Y -111.0989,Z 121,A -108.741,B 24.9567,C -1.5195,E1 24.9585,E2 194.7923} C_DIS
LIN {X -32.1435,Y -110.2307,Z 121,A -110.235,B 24.9564,C -1.5262,E1 24.9545,E2 196.2727} C_DIS
LIN {X -37.0353,Y -108.6842,Z 121,A -112.9055,B 24.9565,C -1.5235,E1 24.9474,E2 198.9544} C_DIS
LIN {X -40.6051,Y -107.4009,Z 121,A -114.7259,B 24.9562,C -1.5284,E1 24.9426,E2 200.7671} C_DIS
LIN {X -43.4906,Y -106.2654,Z 121,A -116.1947,B 24.956,C -1.5332,E1 24.9388,E2 202.2276} C_DIS
LIN {X -46.6095,Y -104.9365,Z 121,A -118.0903,B 24.9563,C -1.5264,E1 24.9339,E2 204.1438} C_DIS
LIN {X -50.5345,Y -103.1031,Z 121,A -120.1881,B 24.956,C -1.5317,E1 24.9287,E2 206.2344} C_DIS
LIN {X -54.6768,Y -100.9662,Z 121,A -122.5184,B 24.9559,C -1.5346,E1 24.9229,E2 208.5642} C_DIS
LIN {X -57.0172,Y -99.6635,Z 121,A -124.0126,B 24.9561,C -1.5299,E1 24.9193,E2 210.0741} C_DIS
LIN {X -61.5644,Y -96.9218,Z 121,A -126.5937,B 24.9558,C -1.5367,E1 24.9131,E2 212.6469} C_DIS
LIN {X -64.739,Y -94.8303,Z 121,A -128.4238,B 24.9554,C -1.5426,E1 24.9089,E2 214.4692} C_DIS
LIN {X -67.6343,Y -92.7868,Z 121,A -130.1608,B 24.9552,C -1.5469,E1 24.905,E2 216.2018} C_DIS
LIN {X -70.4139,Y -90.6961,Z 121,A -132.0179,B 24.9552,C -1.545,E1 24.9008,E2 218.0703} C_DIS
LIN {X -72.6844,Y -88.8873,Z 121,A -133.8012,B 24.9559,C -1.534,E1 24.8969,E2 219.8866} C_DIS
LIN {X -75.3829,Y -86.6094,Z 121,A -135.0954,B 24.9546,C -1.5567,E1 24.8943,E2 221.1319} C_DIS
LIN {X -77.6106,Y -84.6186,Z 121,A -136.4735,B 24.9542,C -1.5643,E1 24.8914,E2 222.4973} C_DIS
LIN {X -81.3309,Y -81.051,Z 121,A -139.2429,B 24.9543,C -1.5616,E1 24.8859,E2 225.2847} C_DIS
LIN {X -83.654,Y -78.6494,Z 121,A -140.9222,B 24.9541,C -1.5648,E1 24.8826,E2 226.9637} C_DIS
LIN {X -86.9379,Y -75.0067,Z 121,A -143.4481,B 24.954,C -1.5671,E1 24.8779,E2 229.4954} C_DIS
LIN {X -89.1948,Y -72.305,Z 121,A -145.5628,B 24.9546,C -1.5568,E1 24.8741,E2 231.6444} C_DIS
LIN {X -91.4848,Y -69.3869,Z 121,A -147.0333,B 24.9534,C -1.5767,E1 24.8717,E2 233.0745} C_DIS
LIN {X -93.561,Y -66.559,Z 121,A -148.6774,B 24.9529,C -1.5855,E1 24.869,E2 234.7058} C_DIS
Enddeposition()
END
